(* CoDeSys 2.3.9.42 project: GLX_VCU_v3.3.0.pro *)
(* Author: JvL *)
(* Libraries: ifm_RAWCan\ifm_RAWCan_NT_V020004.lib 7.6.24 16:48:07, ifm_CR0403\ifm_CR0403_V030400.lib 31.5.24 17:04:27, ifm_CANopen\ifm_NetVarLib_NT_V020004.lib 7.6.24 16:46:42, standard.lib 4.10.05 11:14:46, SysLibCallback.lib 7.6.24 16:43:25, 3S_CANOPENNETVAR.LIB 7.6.24 16:46:41, Iecsfc.lib 13.4.06 15:51:28, Util.lib 7.6.24 16:43:26, ifm_CANopen\3S_CANopenManager.lib 7.6.24 16:46:41, ifm_CANopen\3S_CanDrv.lib 7.6.24 16:46:41 *)

(* PLC configuration (modules and I/O channels)
Configuration [LocalConfiguration] node 0, in %IB0 out %QB0 {IFM_PARAM_WORD_TIME = 0}
AT %IB0 [ChInputBool] Input 00 Bit
AT %IB1 [ChInputBool] Input 01 Bit
AT %IB2 [ChInputBool] Input 02 Bit
AT %IB3 [ChInputBool] Input 03 Bit
IGNITION_KEY AT %IB4 [ChInputBool] Input 04 Bit
CHARGER_INPUT AT %IB5 [ChInputBool] Input 05 Bit
BATTERY1_IGNITION AT %IB6 [ChInputBool] Input 06 Bit
BATTERY2_IGNITION AT %IB7 [ChInputBool] Input 07 Bit
ARM_SWITCH AT %IB8 [ChInputBool] Input 08 Bit
KILL_SWITCH AT %IB9 [ChInputBool] Input 09 Bit
HYDRAULIC_SWITCH AT %IB10 [ChInputBool] Input 10 Bit
EM_SWITCH AT %IB11 [ChInputBool] Input 11 Bit
ARM_LED AT %QB0 [ChOutputBool] Output 00 Bit
PRECHARGE_RELAY AT %QB1 [ChOutputBool] Output 01 Bit
AT %QB2 [ChOutputBool] Output 02 Bit
BRAKE_LIGHT AT %QB3 [ChOutputBool] Output 03 Bit
EM_BRAKE AT %QB4 [ChOutputBool] Output 04 Bit
MCU_IGNITION AT %QB5 [ChOutputBool] Output 05 Bit
BATTERY1_RELAY AT %QB6 [ChOutputBool] Output 06 Bit
BATTERY2_RELAY AT %QB7 [ChOutputBool] Output 07 Bit
HORN AT %QB8 [ChOutputBool] Output 08 Bit
BUZZER AT %QB9 [ChOutputBool] Output 09 Bit
CONTACTOR AT %QB10 [ChOutputBool] Output 10 Bit
CHARGING_LED AT %QB11 [ChOutputBool] Output 11 Bit
System Inputs [LocalSystemInputs] node 2, in %IB12 out %QB12
  SUPPLY_VOLTAGE_VBBS AT %IW6 [ChInputWord] Supply voltage VBBS
  SUPPLY_VOLTAGE_VU AT %IW7 [ChInputWord] Supply voltage VU
  SUPPLY_VOLTAGE_VBB1 AT %IW8 [ChInputWord] Supply voltage VBB1
  SUPPLY_VOLTAGE_VBB2 AT %IW9 [ChInputWord] Supply voltage VBB2
  TEMPERATURE AT %IW10 [ChInputInt] Temperature
J1939 Interface [CAN_J1939] node 1, in %IB37 out %QB12
Interface CAN 2 [CAN_BUS] node 1, in %IB37 out %QB12 {STACK_DWORD_S = 0}
  J1939 Interface [CAN_J1939] node 1, in %IB37 out %QB12
*)

(* Global variable list: CanOpen implicit Variables *)
VAR_GLOBAL CONSTANT
	MAX_CTRLINDEX : INT := 0;
END_VAR

(* Global variable list: Global_Variables *)
VAR_GLOBAL
(*BATTERY*)
	BATTERY1_SOC: BYTE;
	BATTERY1_SOH: BYTE;
	BATTERY1_CHARGING: BOOL;
	BATTERY1_POWER: INT;
	BATTERY1_NTC1: BYTE;
	BATTERY1_NTC2: BYTE;
	BATTERY1_CAN_ERROR: BOOL;
	BATTERY1_CAPACITY: INT;
	BATTERY1_TOTAL_CAPACITY: INT;
	BATTERY1_CURRENT: INT;
	BATTERY1_FULLCHARGE_MIN: REAL;

	BATTERY2_SOC: BYTE;
	BATTERY2_SOH: BYTE;
	BATTERY2_CHARGING: BOOL;
	BATTERY2_POWER: INT;
	BATTERY2_NTC1: BYTE;
	BATTERY2_NTC2: BYTE;
	BATTERY2_CAN_ERROR: BOOL;
	BATTERY2_CAPACITY: INT;
	BATTERY2_TOTAL_CAPACITY: INT;
	BATTERY2_CURRENT: INT;
	BATTERY2_FULLCHARGE_MIN: REAL;

(*MCU <> MOTOR*)
	MOTOR_TARGET_RPM: ARRAY [1..6] OF INT;
	MOTOR_IGNITION: ARRAY [1..6] OF BOOL;

	MOTOR_RPM: ARRAY [1..6] OF INT;
	MOTOR_POWER: ARRAY [1..6] OF INT;
	MOTOR_PHASE_CURRENT: ARRAY [1..6] OF WORD;
	MOTOR_TEMPERATURE:ARRAY [1..6] OF BYTE;
	MCU_TEMPERATURE:ARRAY [1..6] OF BYTE;
	MCU_CAN_ERROR: ARRAY [1..6] OF BOOL;

	MOTOR1_FAULT_ARRAY: ARRAY [1..4] OF BYTE;
	MOTOR2_FAULT_ARRAY: ARRAY [1..4] OF BYTE;
	MOTOR6_FAULT_ARRAY: ARRAY [1..4] OF BYTE;
       MOTOR_OBD_ARRAY: ARRAY [1..6] OF WORD;

(*JOYSTICK*)
	LOG_JX: BYTE;
	LOG_JY: BYTE;
	JOY_ERROR: BOOL;
(*IMU*)
	X_ANGLE_BYTE:BYTE;
	Y_ANGLE_BYTE:BYTE;
	NEG_Y: BOOL;
	NEG_X: BOOL;
	Y_MAX_PEAK: BYTE;
	X_MAX_PEAK: BYTE;
	Y_MIN_PEAK: BYTE;
	X_MIN_PEAK: BYTE;
	IMU_CAN_ERROR:BOOL;
	IMU_ALERT: BOOL;
(*DISPLAY TELEMATICS*)
	HIGH_SPEED: BOOL;
	POWER_MODE: BOOL;
	HILL_HOLD: BOOL;
	DISABLE_MCU_CAN: BOOL;
	TRIP_RESET: BOOL;
      	BATTERY_CHARGING:BOOL;
(*MISC*)
	REVERSE: BOOL;
	MCU_BRAKE: BOOL;
(*HYDRAULICS*)
	HYDRAULIC_IGNITION: BOOL;
(*CALCULATIONS*)
	AVG_RPM: INT;
	RANGE_IN_KM: BYTE;
	SPEED: BYTE;

	RUNTIME: DWORD;
	HYDL_UP_TIME:DWORD;
	VEHICLE_UP_TIME: DWORD;
	VEHICLE_UP_TIME_LT: DWORD;

	ODO_KM: WORD;
	ODO_METER: DWORD;

	TRIP_METER: DWORD;
	TRIP_KM: WORD;

	DUMMY: BOOL;
END_VAR
VAR_GLOBAL RETAIN
	Y_MAX_RETAIN: BYTE;
	X_MAX_RETAIN: BYTE;
	Y_MIN_RETAIN: BYTE;
	X_MIN_RETAIN: BYTE;
END_VAR

(* Global variable list: Networkmanagement implicit Variables CAN *)
VAR_GLOBAL CONSTANT
	USE_NWVARS_CAN : BOOL := FALSE;
	MAX_NetVarItems_CAN	: INT := 0;
	MAX_NetVarPDO_Rx_CAN	: INT := 0;
	MAX_NetVarPDO_Tx_CAN	: INT := 0;
	MAX_NetVarOD_CAN		: INT := 0;
END_VAR
VAR_GLOBAL
	pNetVarItems_CAN		: ARRAY[0..MAX_NetVarItems_CAN] OF NetVarDataItem_CAN;
	pNetVarPDO_Rx_CAN		: ARRAY[0..MAX_NetVarPDO_Rx_CAN] OF NetVarPDO_Rx_CAN;
	pNetVarPDO_Tx_CAN		: ARRAY[0..MAX_NetVarPDO_Tx_CAN] OF NetVarPDO_Tx_CAN;
	pNetVarOD_CAN			: ARRAY[0..MAX_NetVarOD_CAN] OF NetVarOD_CAN;
END_VAR

(* POU PLC_PRG, FBD *)
PROGRAM PLC_PRG
VAR
	CONTACTOR_DELAY: TON;
END_VAR
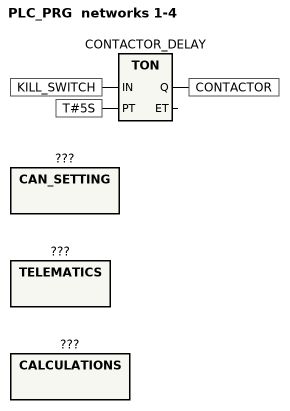
_FBD_ (* Function Block Diagram *)
NETWORK 1
	CONTACTOR_DELAY:TON(IN: KILL_SWITCH, PT: T#5S) => CONTACTOR
NETWORK 2
	???:CAN_SETTING()
NETWORK 3
	???:TELEMATICS()
NETWORK 4
	???:CALCULATIONS()
_END_FBD_
(* the same logic as Structured Text *)
(* Network 1 *)
CONTACTOR_DELAY(IN := KILL_SWITCH, PT := T#5S);
CONTACTOR := CONTACTOR_DELAY.Q;
(* Network 2: see the listing above *)
(* Network 3: see the listing above *)
(* Network 4: see the listing above *)
END_PROGRAM

(* POU CAN_SETTING/CAN_SETTING, FBD *)
PROGRAM CAN_SETTING
(*
Created By: BHAGYESH
Date: 20-01-2024
Version: 1
Description: This program enables the CAN channels and sets the basic CAN parameter for both channels.
This block also controls the IFM's Inbuilt LED.
*)
VAR
	CAN_EN_1: CAN_ENABLE;
	CAN_EN_2: CAN_ENABLE;
	CAN_SET_1: CAN_SETDOWNLOADID;
	CAN_SET_2: CAN_SETDOWNLOADID;
	LED_SET: SET_LED;
	CAN_STATUS_1: CAN_STATUS;
	CAN_STATUS_2: CAN_STATUS;
	RESET_1: BOOL;
	RESET_2: BOOL;
END_VAR
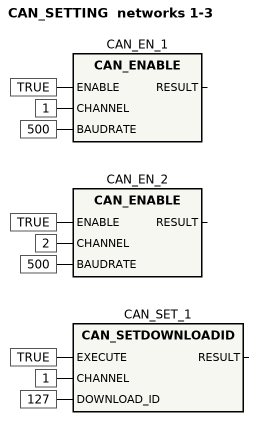
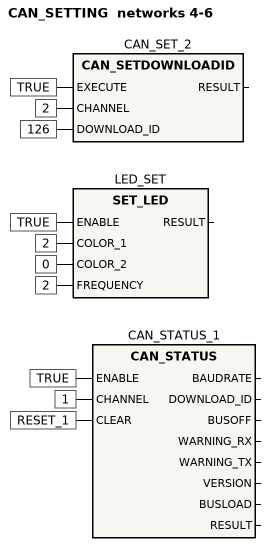
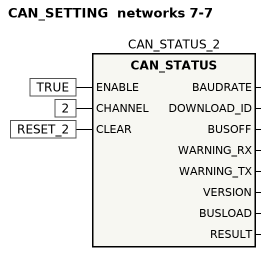
_FBD_ (* Function Block Diagram *)
NETWORK 1
	CAN_EN_1:CAN_ENABLE(ENABLE: TRUE, CHANNEL: 1, BAUDRATE: 500)
NETWORK 2
	CAN_EN_2:CAN_ENABLE(ENABLE: TRUE, CHANNEL: 2, BAUDRATE: 500)
NETWORK 3
	CAN_SET_1:CAN_SETDOWNLOADID(EXECUTE: TRUE, CHANNEL: 1, DOWNLOAD_ID: 127)
NETWORK 4
	CAN_SET_2:CAN_SETDOWNLOADID(EXECUTE: TRUE, CHANNEL: 2, DOWNLOAD_ID: 126)
NETWORK 5
	LED_SET:SET_LED(ENABLE: TRUE, COLOR_1: 2, COLOR_2: 0, FREQUENCY: 2)
NETWORK 6
	CAN_STATUS_1:CAN_STATUS(ENABLE: TRUE, CHANNEL: 1, CLEAR: RESET_1)
NETWORK 7
	CAN_STATUS_2:CAN_STATUS(ENABLE: TRUE, CHANNEL: 2, CLEAR: RESET_2)
_END_FBD_
(* the same logic as Structured Text *)
(* Network 1 *)
CAN_EN_1(ENABLE := TRUE, CHANNEL := 1, BAUDRATE := 500);
(* Network 2 *)
CAN_EN_2(ENABLE := TRUE, CHANNEL := 2, BAUDRATE := 500);
(* Network 3 *)
CAN_SET_1(EXECUTE := TRUE, CHANNEL := 1, DOWNLOAD_ID := 127);
(* Network 4 *)
CAN_SET_2(EXECUTE := TRUE, CHANNEL := 2, DOWNLOAD_ID := 126);
(* Network 5 *)
LED_SET(ENABLE := TRUE, COLOR_1 := 2, COLOR_2 := 0, FREQUENCY := 2);
(* Network 6 *)
CAN_STATUS_1(ENABLE := TRUE, CHANNEL := 1, CLEAR := RESET_1);
(* Network 7 *)
CAN_STATUS_2(ENABLE := TRUE, CHANNEL := 2, CLEAR := RESET_2);
END_PROGRAM

(* POU TELEMATICS, LD *)
PROGRAM TELEMATICS
VAR
	TX_300: CAN_TX;
	TX_301: CAN_TX;
	TX_303: CAN_TX;
	TX_305: CAN_TX;
	TX_306: CAN_TX;
   	TX_307: CAN_TX;
	TX_308: CAN_TX;
	TX_310: CAN_TX;
	TX_311: CAN_TX;
	TX_312: CAN_TX;
	TX_313: CAN_TX;
	TX_31A: CAN_TX;
	TX_31B: CAN_TX;

	TX_400: CAN_TX;
	TX_401: CAN_TX;
	TX_403: CAN_TX;
	TX_405: CAN_TX;
	TX_406: CAN_TX;
   	TX_407: CAN_TX;
	TX_408: CAN_TX;
	TX_410: CAN_TX;
	TX_411: CAN_TX;
	TX_412: CAN_TX;
	TX_413: CAN_TX;
	TX_41A: CAN_TX;
	TX_41B: CAN_TX;
	TX_262: CAN_TX;

	RX_7F0: RX_CAN;
	RX_450: RX_CAN;

	PACK_301: PACK_BYTES;
	PACK_303: PACK_BYTES;
	PACK_305: PACK_BYTES;
	PACK_306: PACK_BYTES;
	PACK_308: PACK_BYTES;
	PACK_311: PACK_BYTES;
	PACK_313: PACK_BYTES;
	PACK_31B: PACK_BYTES;
	PACK_262: PACK_BYTES;

	WB_BATTERY1_POWER: WORD_BYTE_CONVERSION;
	WB_RPM_1: WORD_BYTE_CONVERSION;
	WB_POWER_1: WORD_BYTE_CONVERSION;
	WB_PHASE_1: WORD_BYTE_CONVERSION;
	WB_TARGET_RPM_1: WORD_BYTE_CONVERSION;

	WB_BATTERY2_POWER: WORD_BYTE_CONVERSION;
	WB_RPM_2: WORD_BYTE_CONVERSION;
	WB_POWER_2: WORD_BYTE_CONVERSION;
	WB_PHASE_2: WORD_BYTE_CONVERSION;
	WB_TARGET_RPM_2: WORD_BYTE_CONVERSION;

	WB_RPM_6: WORD_BYTE_CONVERSION;
	WB_POWER_6: WORD_BYTE_CONVERSION;
	WB_PHASE_6: WORD_BYTE_CONVERSION;
	WB_TARGET_RPM_6: WORD_BYTE_CONVERSION;
	WB_FAULTS_6: WORD_BYTE_CONVERSION;

	WB_RUNTIME: WORD_BYTE_CONVERSION;

	DATA_LOG_ERROR: BOOL;
	DWIN_CAN_ERROR: BOOL;
	TIMER_DATALOG: TON;
	TIMER_DWIN: TON;
	TIMER_TX: TON;

	WD_BATTERY1_FULLCHARGE_MIN: WORD;
	WD_BATTERY2_FULLCHARGE_MIN: WORD;
	WB_FULLCHARGE1_MIN: WORD_BYTE_CONVERSION;
	WB_FULLCHARGE2_MIN: WORD_BYTE_CONVERSION;

	WB_OBD_1: WORD_BYTE_CONVERSION;
	WB_OBD_2: WORD_BYTE_CONVERSION;
	WB_OBD_6: WORD_BYTE_CONVERSION;

	WB_HYDL_UP_TIME: WORD_BYTE_CONVERSION;
	WB_TRIP_KM: WORD_BYTE_CONVERSION;
	WB_ODO_METERS: DWORD_BYTE_CONVERSION;
	WB_RUNTIME_MIN: DWORD_BYTE_CONVERSION;
	TIMER_TX_1: TON;
	TIMER_TX_2: TON;
	RX_3A0: RX_CAN;
	TRIP: WORD_BYTE_CONVERSION;
	OBD1_INT: INT;
	OBD1_BYTE: BYTE;
	OBD2_INT: INT;
	OBD2_BYTE: BYTE;
	OBD6_INT: INT;
	OBD6_BYTE: BYTE;
	WB_HYDL_UPTIME: DWORD_BYTE_CONVERSION;
	WB_VEHICLE_UPTIME: DWORD_BYTE_CONVERSION;
	TX_409: CAN_TX;
	PACK_409: PACK_BYTES;
	WB_VEHICLE_UPTIME_LT: DWORD_BYTE_CONVERSION;
END_VAR
VAR CONSTANT
	META_FRAME: ARRAY [0..7] OF BYTE := 18,1,1,0,0,0,0,0; (*GLX_PR, KEY1, VX,VY,VZ*)
	CAN_CHANNEL: BYTE := 1;
END_VAR
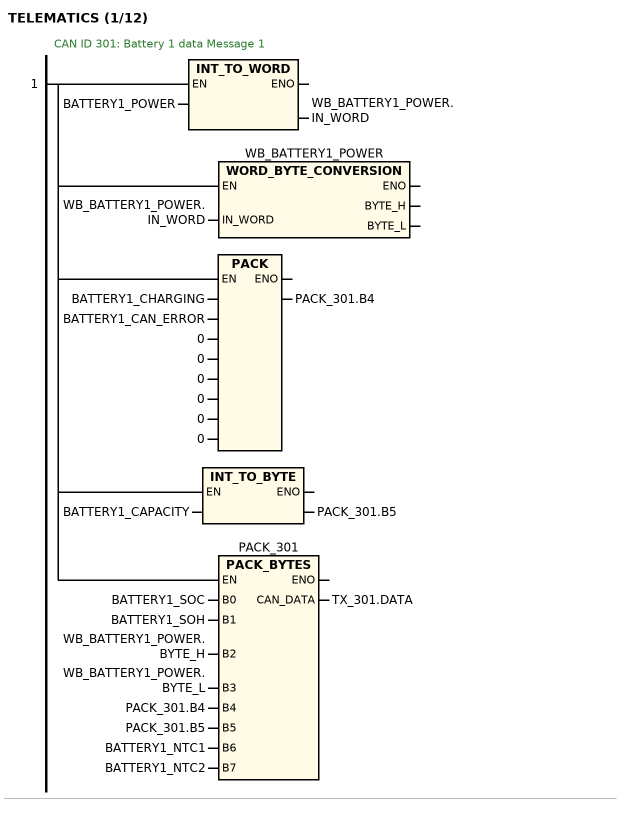
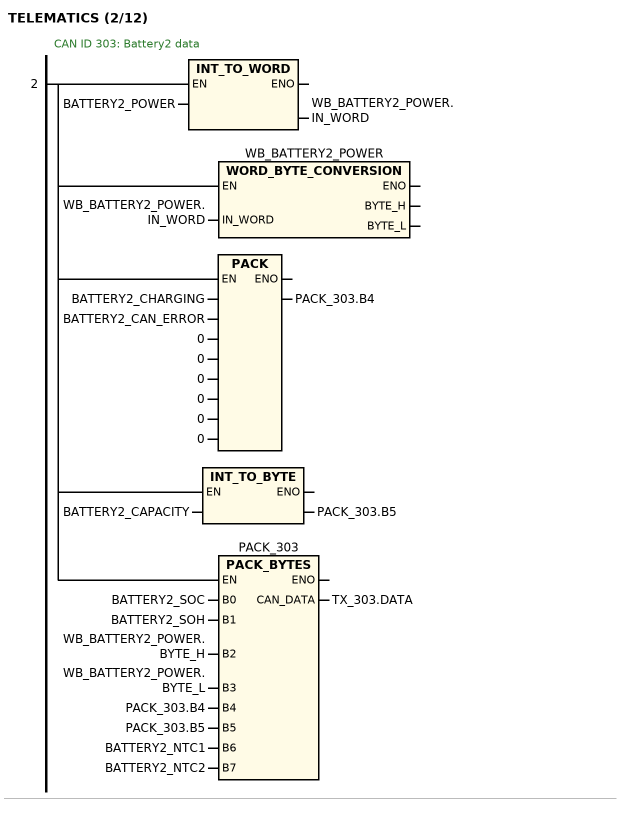
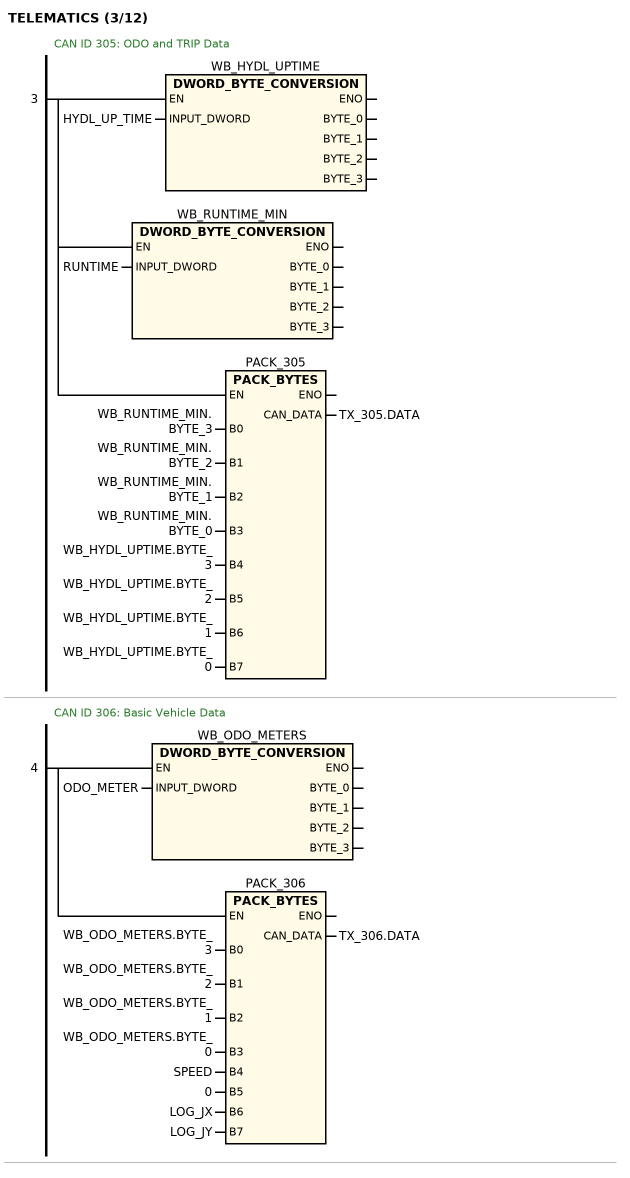
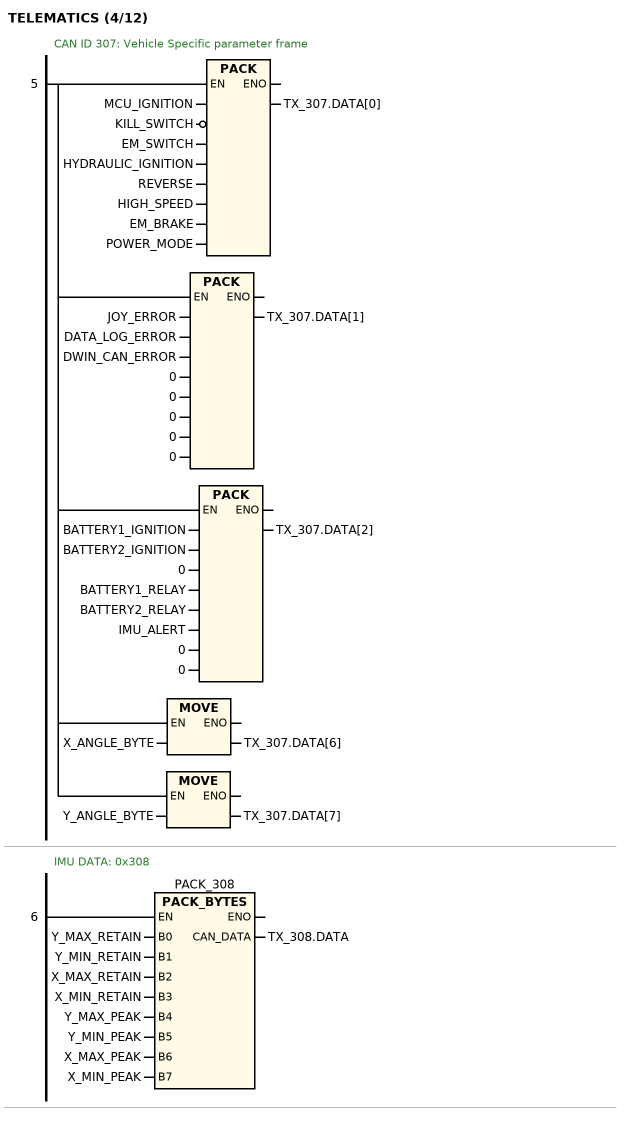
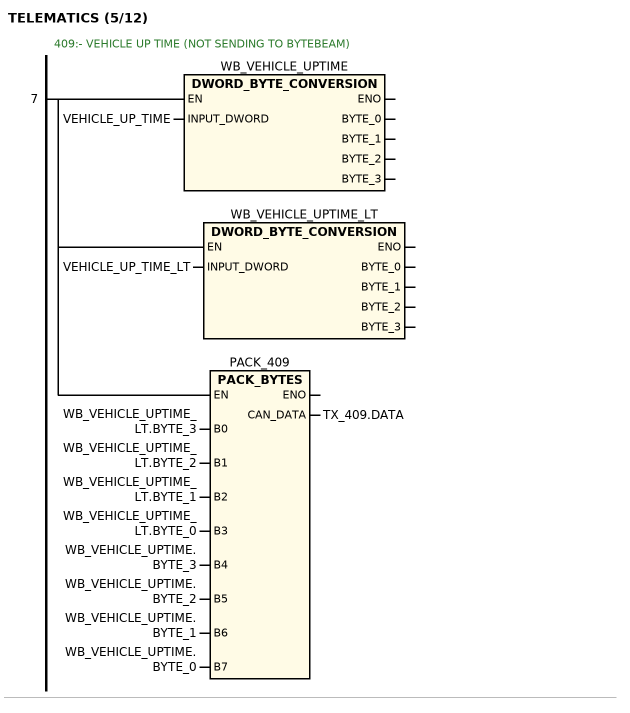
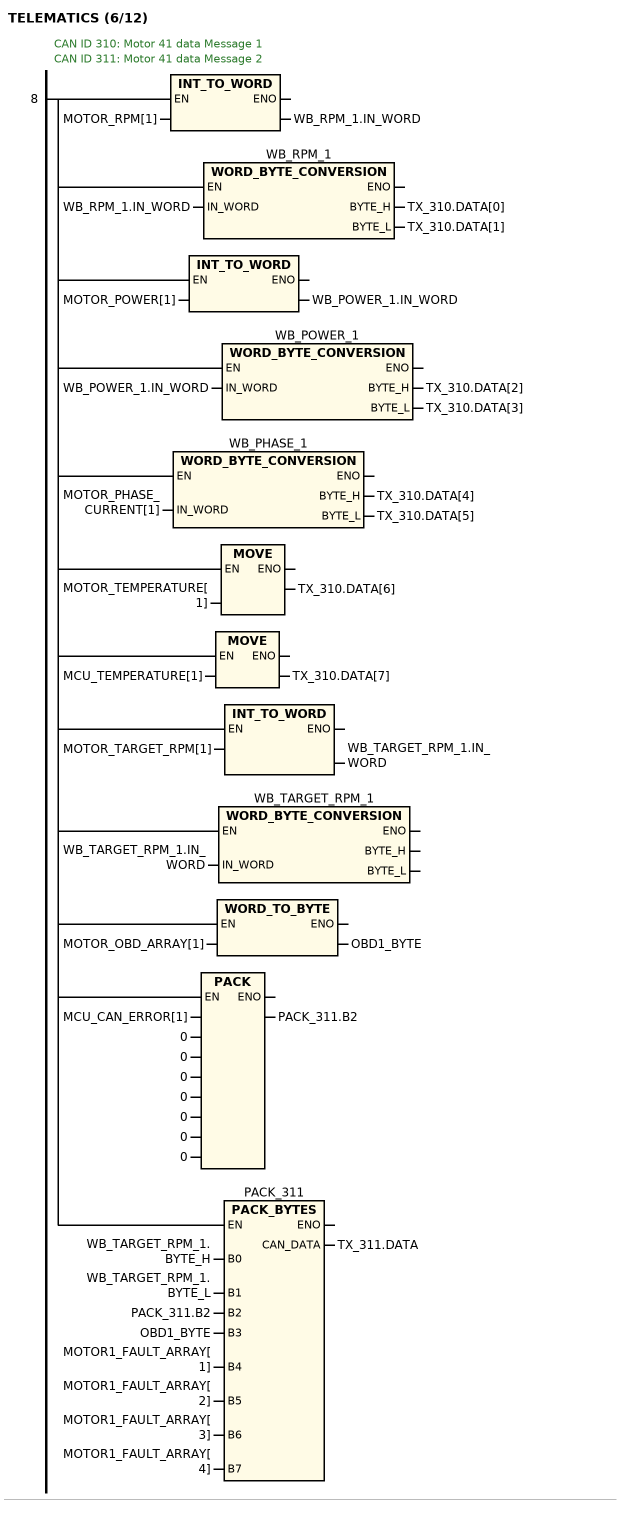
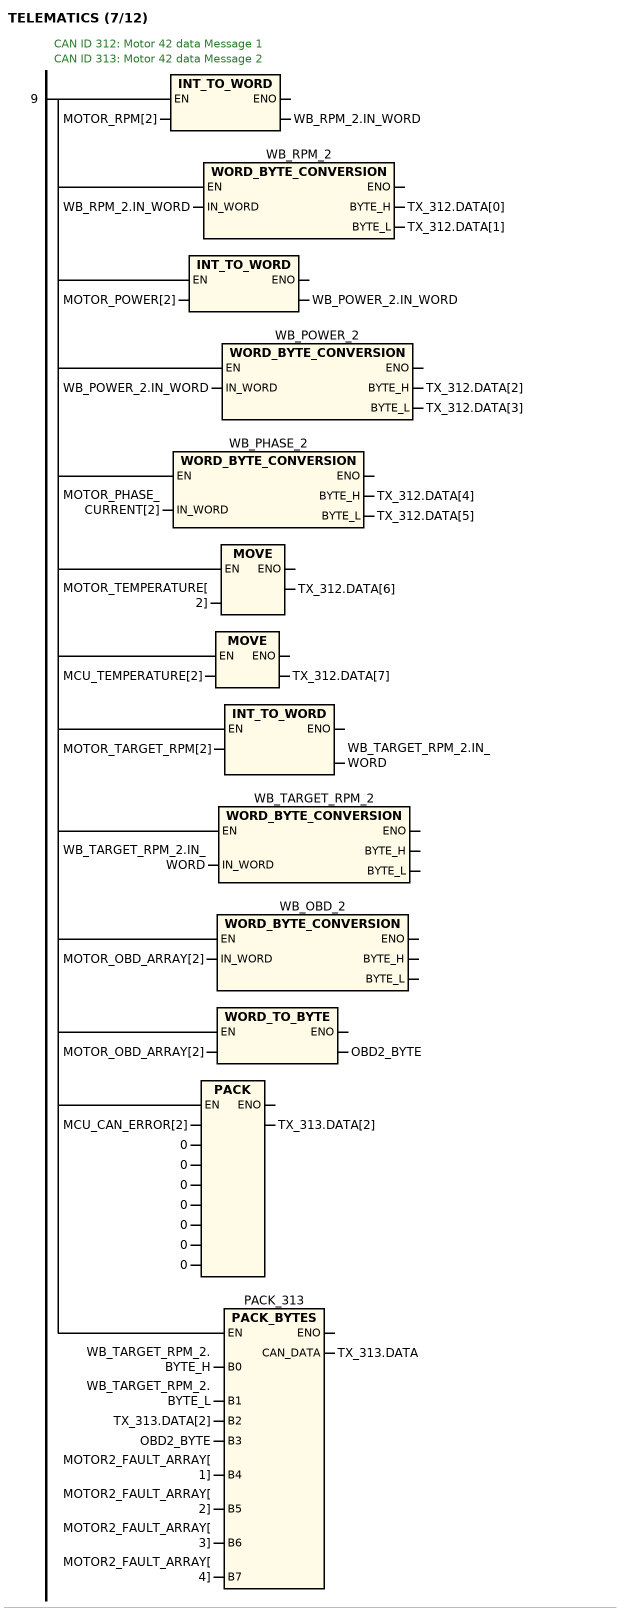
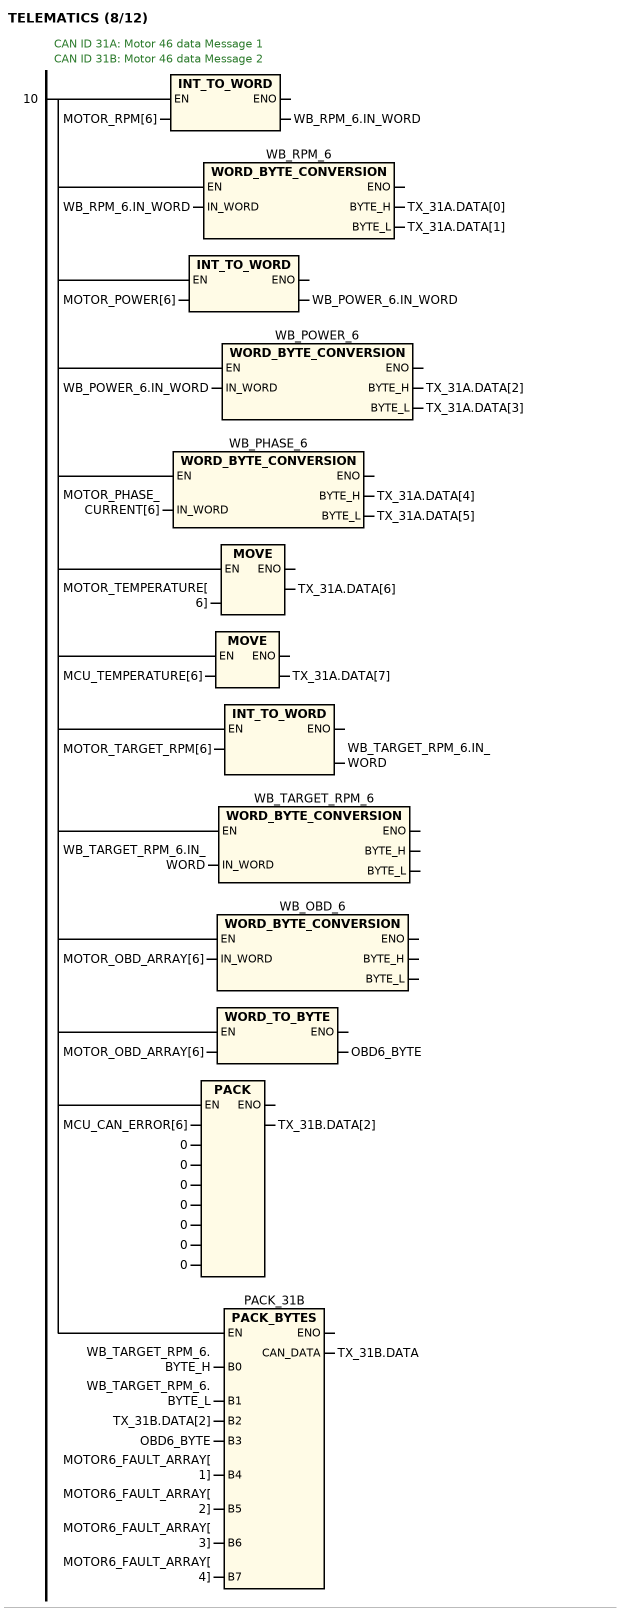
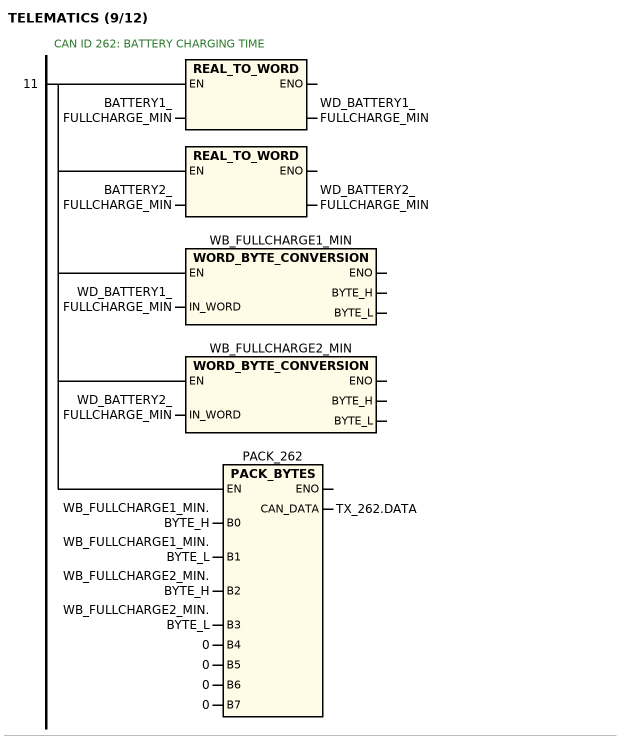
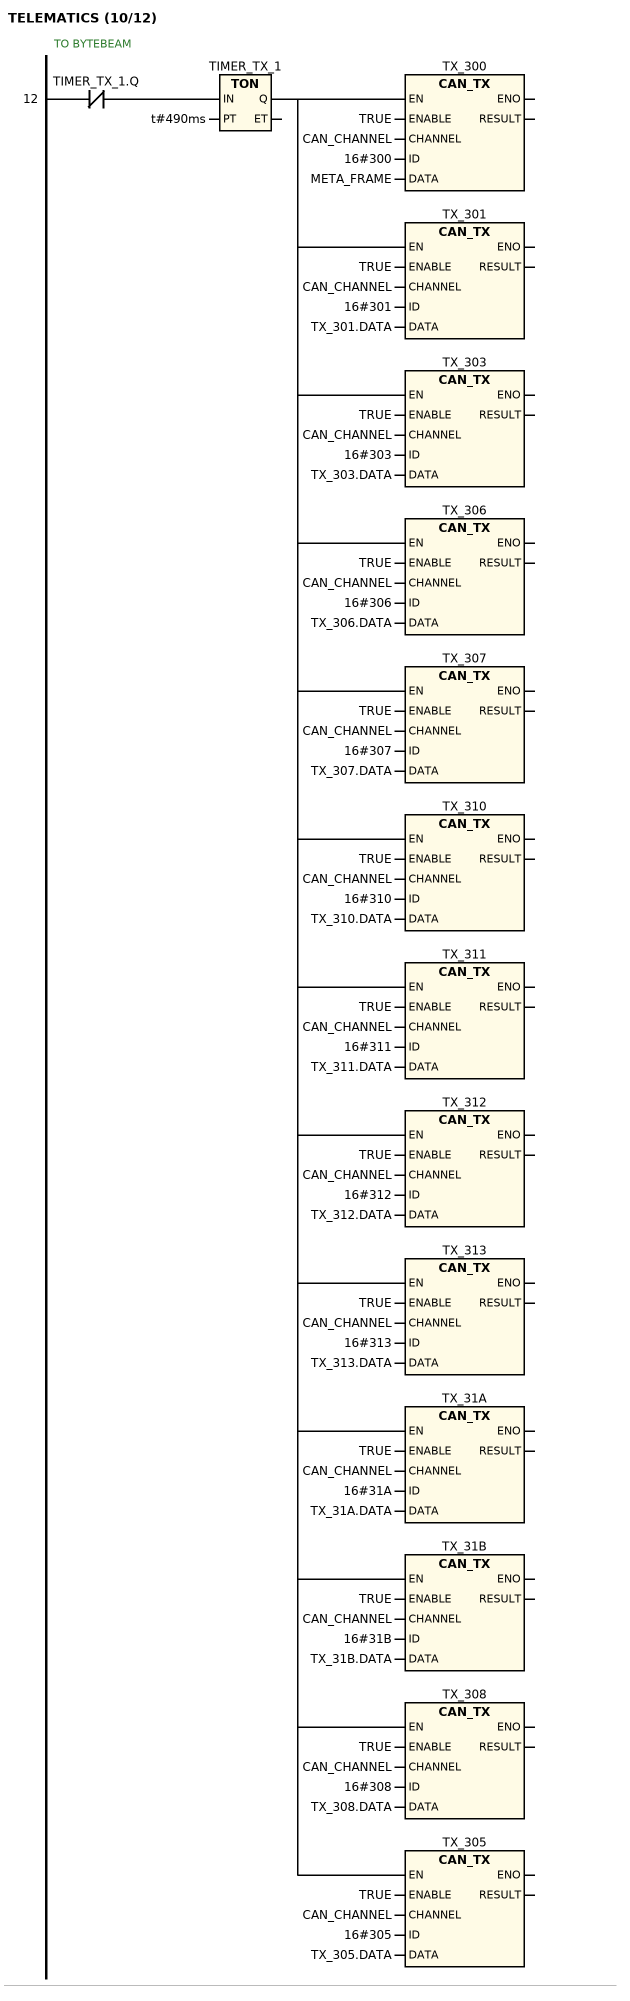
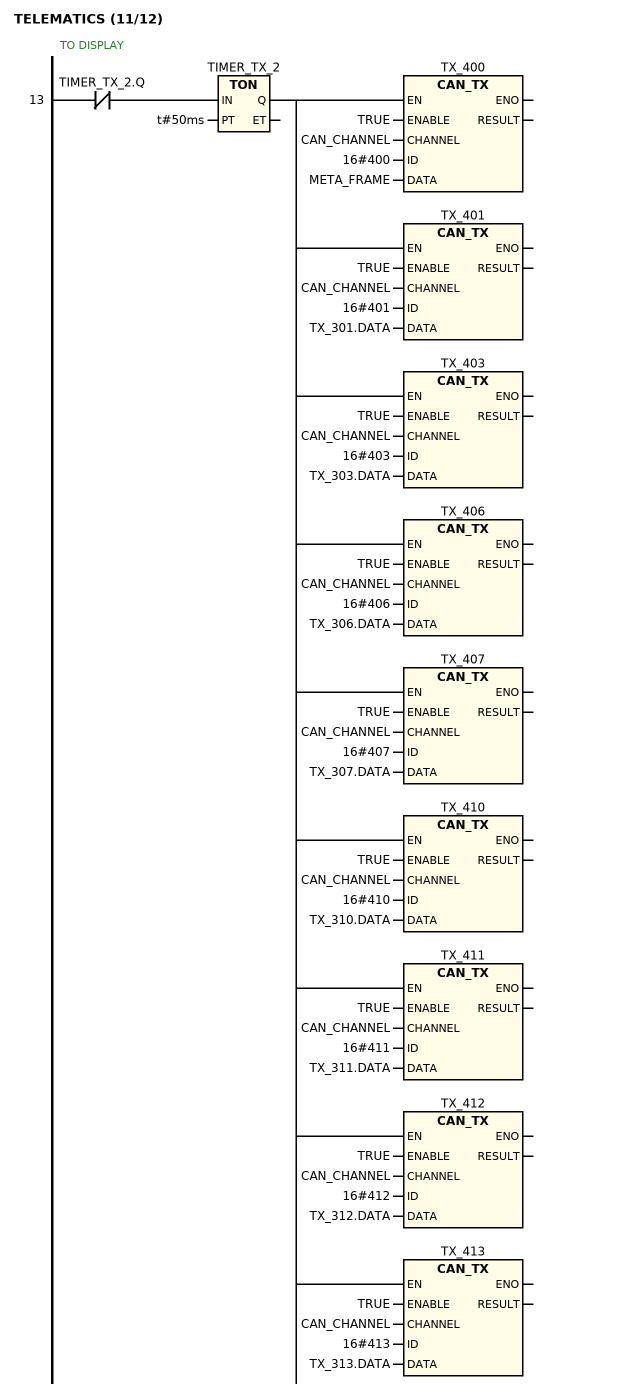
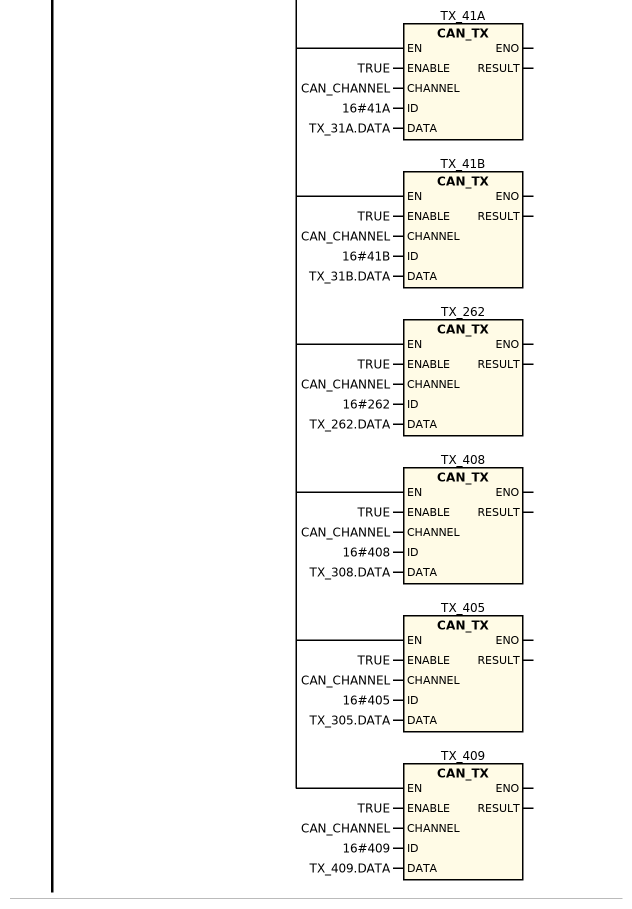
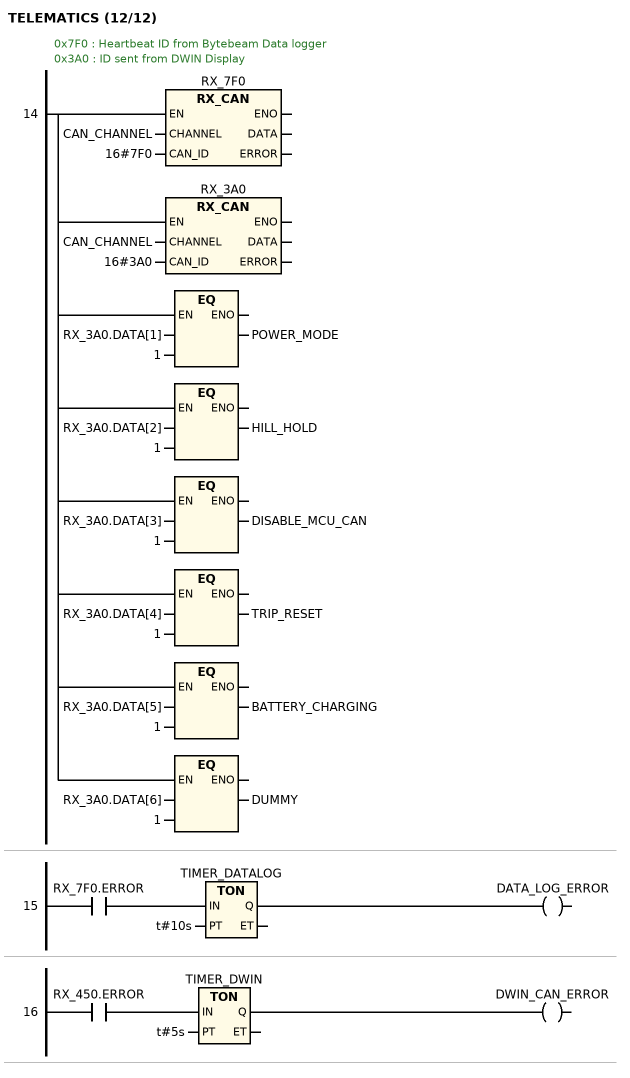
_LD_ (* Ladder Diagram *)
NETWORK 1 (* CAN ID 301: Battery 1 data Message 1 *)
	*
		EN --- INT_TO_WORD(BATTERY1_POWER) => WB_BATTERY1_POWER.IN_WORD
		EN --- WB_BATTERY1_POWER:WORD_BYTE_CONVERSION(IN_WORD: WB_BATTERY1_POWER.IN_WORD)
		EN --- PACK(BATTERY1_CHARGING, BATTERY1_CAN_ERROR, 0, 0, 0, 0, 0, 0) => PACK_301.B4
		EN --- INT_TO_BYTE(BATTERY1_CAPACITY) => PACK_301.B5
		EN --- PACK_301:PACK_BYTES(B0: BATTERY1_SOC, B1: BATTERY1_SOH, B2: WB_BATTERY1_POWER.BYTE_H, B3: WB_BATTERY1_POWER.BYTE_L, B4: PACK_301.B4, B5: PACK_301.B5, B6: BATTERY1_NTC1, B7: BATTERY1_NTC2) => TX_301.DATA
NETWORK 2 (* CAN ID 303: Battery2 data *)
	*
		EN --- INT_TO_WORD(BATTERY2_POWER) => WB_BATTERY2_POWER.IN_WORD
		EN --- WB_BATTERY2_POWER:WORD_BYTE_CONVERSION(IN_WORD: WB_BATTERY2_POWER.IN_WORD)
		EN --- PACK(BATTERY2_CHARGING, BATTERY2_CAN_ERROR, 0, 0, 0, 0, 0, 0) => PACK_303.B4
		EN --- INT_TO_BYTE(BATTERY2_CAPACITY) => PACK_303.B5
		EN --- PACK_303:PACK_BYTES(B0: BATTERY2_SOC, B1: BATTERY2_SOH, B2: WB_BATTERY2_POWER.BYTE_H, B3: WB_BATTERY2_POWER.BYTE_L, B4: PACK_303.B4, B5: PACK_303.B5, B6: BATTERY2_NTC1, B7: BATTERY2_NTC2) => TX_303.DATA
NETWORK 3 (* CAN ID 305: ODO and TRIP Data *)
	*
		EN --- WB_HYDL_UPTIME:DWORD_BYTE_CONVERSION(INPUT_DWORD: HYDL_UP_TIME)
		EN --- WB_RUNTIME_MIN:DWORD_BYTE_CONVERSION(INPUT_DWORD: RUNTIME)
		EN --- PACK_305:PACK_BYTES(B0: WB_RUNTIME_MIN.BYTE_3, B1: WB_RUNTIME_MIN.BYTE_2, B2: WB_RUNTIME_MIN.BYTE_1, B3: WB_RUNTIME_MIN.BYTE_0, B4: WB_HYDL_UPTIME.BYTE_3, B5: WB_HYDL_UPTIME.BYTE_2, B6: WB_HYDL_UPTIME.BYTE_1, B7: WB_HYDL_UPTIME.BYTE_0) => TX_305.DATA
NETWORK 4 (* CAN ID 306: Basic Vehicle Data *)
	*
		EN --- WB_ODO_METERS:DWORD_BYTE_CONVERSION(INPUT_DWORD: ODO_METER)
		EN --- PACK_306:PACK_BYTES(B0: WB_ODO_METERS.BYTE_3, B1: WB_ODO_METERS.BYTE_2, B2: WB_ODO_METERS.BYTE_1, B3: WB_ODO_METERS.BYTE_0, B4: SPEED, B5: 0, B6: LOG_JX, B7: LOG_JY) => TX_306.DATA
NETWORK 5 (* CAN ID 307: Vehicle Specific parameter frame *)
	*
		EN --- PACK(MCU_IGNITION, NOT KILL_SWITCH, EM_SWITCH, HYDRAULIC_IGNITION, REVERSE, HIGH_SPEED, EM_BRAKE, POWER_MODE) => TX_307.DATA[0]
		EN --- PACK(JOY_ERROR, DATA_LOG_ERROR, DWIN_CAN_ERROR, 0, 0, 0, 0, 0) => TX_307.DATA[1]
		EN --- PACK(BATTERY1_IGNITION, BATTERY2_IGNITION, 0, BATTERY1_RELAY, BATTERY2_RELAY, IMU_ALERT, 0, 0) => TX_307.DATA[2]
		EN --- MOVE(X_ANGLE_BYTE) => TX_307.DATA[6]
		EN --- MOVE(Y_ANGLE_BYTE) => TX_307.DATA[7]
NETWORK 6 (* IMU DATA: 0x308 *)
	*
		EN --- PACK_308:PACK_BYTES(B0: Y_MAX_RETAIN, B1: Y_MIN_RETAIN, B2: X_MAX_RETAIN, B3: X_MIN_RETAIN, B4: Y_MAX_PEAK, B5: Y_MIN_PEAK, B6: X_MAX_PEAK, B7: X_MIN_PEAK) => TX_308.DATA
NETWORK 7 (* 409:- VEHICLE UP TIME (NOT SENDING TO BYTEBEAM) *)
	*
		EN --- WB_VEHICLE_UPTIME:DWORD_BYTE_CONVERSION(INPUT_DWORD: VEHICLE_UP_TIME)
		EN --- WB_VEHICLE_UPTIME_LT:DWORD_BYTE_CONVERSION(INPUT_DWORD: VEHICLE_UP_TIME_LT)
		EN --- PACK_409:PACK_BYTES(B0: WB_VEHICLE_UPTIME_LT.BYTE_3, B1: WB_VEHICLE_UPTIME_LT.BYTE_2, B2: WB_VEHICLE_UPTIME_LT.BYTE_1, B3: WB_VEHICLE_UPTIME_LT.BYTE_0, B4: WB_VEHICLE_UPTIME.BYTE_3, B5: WB_VEHICLE_UPTIME.BYTE_2, B6: WB_VEHICLE_UPTIME.BYTE_1, B7: WB_VEHICLE_UPTIME.BYTE_0) => TX_409.DATA
NETWORK 8 (* CAN ID 310: Motor 41 data Message 1 / CAN ID 311: Motor 41 data Message 2 *)
	*
		EN --- INT_TO_WORD(MOTOR_RPM[1]) => WB_RPM_1.IN_WORD
		EN --- WB_RPM_1:WORD_BYTE_CONVERSION(IN_WORD: WB_RPM_1.IN_WORD, BYTE_L => TX_310.DATA[1]) => TX_310.DATA[0]
		EN --- INT_TO_WORD(MOTOR_POWER[1]) => WB_POWER_1.IN_WORD
		EN --- WB_POWER_1:WORD_BYTE_CONVERSION(IN_WORD: WB_POWER_1.IN_WORD, BYTE_L => TX_310.DATA[3]) => TX_310.DATA[2]
		EN --- WB_PHASE_1:WORD_BYTE_CONVERSION(IN_WORD: MOTOR_PHASE_CURRENT[1], BYTE_L => TX_310.DATA[5]) => TX_310.DATA[4]
		EN --- MOVE(MOTOR_TEMPERATURE[1]) => TX_310.DATA[6]
		EN --- MOVE(MCU_TEMPERATURE[1]) => TX_310.DATA[7]
		EN --- INT_TO_WORD(MOTOR_TARGET_RPM[1]) => WB_TARGET_RPM_1.IN_WORD
		EN --- WB_TARGET_RPM_1:WORD_BYTE_CONVERSION(IN_WORD: WB_TARGET_RPM_1.IN_WORD)
		EN --- WORD_TO_BYTE(MOTOR_OBD_ARRAY[1]) => OBD1_BYTE
		EN --- PACK(MCU_CAN_ERROR[1], 0, 0, 0, 0, 0, 0, 0) => PACK_311.B2
		EN --- PACK_311:PACK_BYTES(B0: WB_TARGET_RPM_1.BYTE_H, B1: WB_TARGET_RPM_1.BYTE_L, B2: PACK_311.B2, B3: OBD1_BYTE, B4: MOTOR1_FAULT_ARRAY[1], B5: MOTOR1_FAULT_ARRAY[2], B6: MOTOR1_FAULT_ARRAY[3], B7: MOTOR1_FAULT_ARRAY[4]) => TX_311.DATA
NETWORK 9 (* CAN ID 312: Motor 42 data Message 1 / CAN ID 313: Motor 42 data Message 2 *)
	*
		EN --- INT_TO_WORD(MOTOR_RPM[2]) => WB_RPM_2.IN_WORD
		EN --- WB_RPM_2:WORD_BYTE_CONVERSION(IN_WORD: WB_RPM_2.IN_WORD, BYTE_L => TX_312.DATA[1]) => TX_312.DATA[0]
		EN --- INT_TO_WORD(MOTOR_POWER[2]) => WB_POWER_2.IN_WORD
		EN --- WB_POWER_2:WORD_BYTE_CONVERSION(IN_WORD: WB_POWER_2.IN_WORD, BYTE_L => TX_312.DATA[3]) => TX_312.DATA[2]
		EN --- WB_PHASE_2:WORD_BYTE_CONVERSION(IN_WORD: MOTOR_PHASE_CURRENT[2], BYTE_L => TX_312.DATA[5]) => TX_312.DATA[4]
		EN --- MOVE(MOTOR_TEMPERATURE[2]) => TX_312.DATA[6]
		EN --- MOVE(MCU_TEMPERATURE[2]) => TX_312.DATA[7]
		EN --- INT_TO_WORD(MOTOR_TARGET_RPM[2]) => WB_TARGET_RPM_2.IN_WORD
		EN --- WB_TARGET_RPM_2:WORD_BYTE_CONVERSION(IN_WORD: WB_TARGET_RPM_2.IN_WORD)
		EN --- WB_OBD_2:WORD_BYTE_CONVERSION(IN_WORD: MOTOR_OBD_ARRAY[2])
		EN --- WORD_TO_BYTE(MOTOR_OBD_ARRAY[2]) => OBD2_BYTE
		EN --- PACK(MCU_CAN_ERROR[2], 0, 0, 0, 0, 0, 0, 0) => TX_313.DATA[2]
		EN --- PACK_313:PACK_BYTES(B0: WB_TARGET_RPM_2.BYTE_H, B1: WB_TARGET_RPM_2.BYTE_L, B2: TX_313.DATA[2], B3: OBD2_BYTE, B4: MOTOR2_FAULT_ARRAY[1], B5: MOTOR2_FAULT_ARRAY[2], B6: MOTOR2_FAULT_ARRAY[3], B7: MOTOR2_FAULT_ARRAY[4]) => TX_313.DATA
NETWORK 10 (* CAN ID 31A: Motor 46 data Message 1 / CAN ID 31B: Motor 46 data Message 2 *)
	*
		EN --- INT_TO_WORD(MOTOR_RPM[6]) => WB_RPM_6.IN_WORD
		EN --- WB_RPM_6:WORD_BYTE_CONVERSION(IN_WORD: WB_RPM_6.IN_WORD, BYTE_L => TX_31A.DATA[1]) => TX_31A.DATA[0]
		EN --- INT_TO_WORD(MOTOR_POWER[6]) => WB_POWER_6.IN_WORD
		EN --- WB_POWER_6:WORD_BYTE_CONVERSION(IN_WORD: WB_POWER_6.IN_WORD, BYTE_L => TX_31A.DATA[3]) => TX_31A.DATA[2]
		EN --- WB_PHASE_6:WORD_BYTE_CONVERSION(IN_WORD: MOTOR_PHASE_CURRENT[6], BYTE_L => TX_31A.DATA[5]) => TX_31A.DATA[4]
		EN --- MOVE(MOTOR_TEMPERATURE[6]) => TX_31A.DATA[6]
		EN --- MOVE(MCU_TEMPERATURE[6]) => TX_31A.DATA[7]
		EN --- INT_TO_WORD(MOTOR_TARGET_RPM[6]) => WB_TARGET_RPM_6.IN_WORD
		EN --- WB_TARGET_RPM_6:WORD_BYTE_CONVERSION(IN_WORD: WB_TARGET_RPM_6.IN_WORD)
		EN --- WB_OBD_6:WORD_BYTE_CONVERSION(IN_WORD: MOTOR_OBD_ARRAY[6])
		EN --- WORD_TO_BYTE(MOTOR_OBD_ARRAY[6]) => OBD6_BYTE
		EN --- PACK(MCU_CAN_ERROR[6], 0, 0, 0, 0, 0, 0, 0) => TX_31B.DATA[2]
		EN --- PACK_31B:PACK_BYTES(B0: WB_TARGET_RPM_6.BYTE_H, B1: WB_TARGET_RPM_6.BYTE_L, B2: TX_31B.DATA[2], B3: OBD6_BYTE, B4: MOTOR6_FAULT_ARRAY[1], B5: MOTOR6_FAULT_ARRAY[2], B6: MOTOR6_FAULT_ARRAY[3], B7: MOTOR6_FAULT_ARRAY[4]) => TX_31B.DATA
NETWORK 11 (* CAN ID 262: BATTERY CHARGING TIME *)
	*
		EN --- REAL_TO_WORD(BATTERY1_FULLCHARGE_MIN) => WD_BATTERY1_FULLCHARGE_MIN
		EN --- REAL_TO_WORD(BATTERY2_FULLCHARGE_MIN) => WD_BATTERY2_FULLCHARGE_MIN
		EN --- WB_FULLCHARGE1_MIN:WORD_BYTE_CONVERSION(IN_WORD: WD_BATTERY1_FULLCHARGE_MIN)
		EN --- WB_FULLCHARGE2_MIN:WORD_BYTE_CONVERSION(IN_WORD: WD_BATTERY2_FULLCHARGE_MIN)
		EN --- PACK_262:PACK_BYTES(B0: WB_FULLCHARGE1_MIN.BYTE_H, B1: WB_FULLCHARGE1_MIN.BYTE_L, B2: WB_FULLCHARGE2_MIN.BYTE_H, B3: WB_FULLCHARGE2_MIN.BYTE_L, B4: 0, B5: 0, B6: 0, B7: 0) => TX_262.DATA
NETWORK 12 (* TO BYTEBEAM *)
	[/TIMER_TX_1.Q] - TIMER_TX_1:TON(IN: *, PT: t#490ms)
		EN --- TX_300:CAN_TX(ENABLE: TRUE, CHANNEL: CAN_CHANNEL, ID: 16#300, DATA: META_FRAME)
		EN --- TX_301:CAN_TX(ENABLE: TRUE, CHANNEL: CAN_CHANNEL, ID: 16#301, DATA: TX_301.DATA)
		EN --- TX_303:CAN_TX(ENABLE: TRUE, CHANNEL: CAN_CHANNEL, ID: 16#303, DATA: TX_303.DATA)
		EN --- TX_306:CAN_TX(ENABLE: TRUE, CHANNEL: CAN_CHANNEL, ID: 16#306, DATA: TX_306.DATA)
		EN --- TX_307:CAN_TX(ENABLE: TRUE, CHANNEL: CAN_CHANNEL, ID: 16#307, DATA: TX_307.DATA)
		EN --- TX_310:CAN_TX(ENABLE: TRUE, CHANNEL: CAN_CHANNEL, ID: 16#310, DATA: TX_310.DATA)
		EN --- TX_311:CAN_TX(ENABLE: TRUE, CHANNEL: CAN_CHANNEL, ID: 16#311, DATA: TX_311.DATA)
		EN --- TX_312:CAN_TX(ENABLE: TRUE, CHANNEL: CAN_CHANNEL, ID: 16#312, DATA: TX_312.DATA)
		EN --- TX_313:CAN_TX(ENABLE: TRUE, CHANNEL: CAN_CHANNEL, ID: 16#313, DATA: TX_313.DATA)
		EN --- TX_31A:CAN_TX(ENABLE: TRUE, CHANNEL: CAN_CHANNEL, ID: 16#31A, DATA: TX_31A.DATA)
		EN --- TX_31B:CAN_TX(ENABLE: TRUE, CHANNEL: CAN_CHANNEL, ID: 16#31B, DATA: TX_31B.DATA)
		EN --- TX_308:CAN_TX(ENABLE: TRUE, CHANNEL: CAN_CHANNEL, ID: 16#308, DATA: TX_308.DATA)
		EN --- TX_305:CAN_TX(ENABLE: TRUE, CHANNEL: CAN_CHANNEL, ID: 16#305, DATA: TX_305.DATA)
NETWORK 13 (* TO DISPLAY *)
	[/TIMER_TX_2.Q] - TIMER_TX_2:TON(IN: *, PT: t#50ms)
		EN --- TX_400:CAN_TX(ENABLE: TRUE, CHANNEL: CAN_CHANNEL, ID: 16#400, DATA: META_FRAME)
		EN --- TX_401:CAN_TX(ENABLE: TRUE, CHANNEL: CAN_CHANNEL, ID: 16#401, DATA: TX_301.DATA)
		EN --- TX_403:CAN_TX(ENABLE: TRUE, CHANNEL: CAN_CHANNEL, ID: 16#403, DATA: TX_303.DATA)
		EN --- TX_406:CAN_TX(ENABLE: TRUE, CHANNEL: CAN_CHANNEL, ID: 16#406, DATA: TX_306.DATA)
		EN --- TX_407:CAN_TX(ENABLE: TRUE, CHANNEL: CAN_CHANNEL, ID: 16#407, DATA: TX_307.DATA)
		EN --- TX_410:CAN_TX(ENABLE: TRUE, CHANNEL: CAN_CHANNEL, ID: 16#410, DATA: TX_310.DATA)
		EN --- TX_411:CAN_TX(ENABLE: TRUE, CHANNEL: CAN_CHANNEL, ID: 16#411, DATA: TX_311.DATA)
		EN --- TX_412:CAN_TX(ENABLE: TRUE, CHANNEL: CAN_CHANNEL, ID: 16#412, DATA: TX_312.DATA)
		EN --- TX_413:CAN_TX(ENABLE: TRUE, CHANNEL: CAN_CHANNEL, ID: 16#413, DATA: TX_313.DATA)
		EN --- TX_41A:CAN_TX(ENABLE: TRUE, CHANNEL: CAN_CHANNEL, ID: 16#41A, DATA: TX_31A.DATA)
		EN --- TX_41B:CAN_TX(ENABLE: TRUE, CHANNEL: CAN_CHANNEL, ID: 16#41B, DATA: TX_31B.DATA)
		EN --- TX_262:CAN_TX(ENABLE: TRUE, CHANNEL: CAN_CHANNEL, ID: 16#262, DATA: TX_262.DATA)
		EN --- TX_408:CAN_TX(ENABLE: TRUE, CHANNEL: CAN_CHANNEL, ID: 16#408, DATA: TX_308.DATA)
		EN --- TX_405:CAN_TX(ENABLE: TRUE, CHANNEL: CAN_CHANNEL, ID: 16#405, DATA: TX_305.DATA)
		EN --- TX_409:CAN_TX(ENABLE: TRUE, CHANNEL: CAN_CHANNEL, ID: 16#409, DATA: TX_409.DATA)
NETWORK 14 (* 0x7F0 : Heartbeat ID from Bytebeam Data logger / 0x3A0 : ID sent from DWIN Display *)
	*
		EN --- RX_7F0:RX_CAN(CHANNEL: CAN_CHANNEL, CAN_ID: 16#7F0)
		EN --- RX_3A0:RX_CAN(CHANNEL: CAN_CHANNEL, CAN_ID: 16#3A0)
		EN --- EQ(RX_3A0.DATA[1], 1) => POWER_MODE
		EN --- EQ(RX_3A0.DATA[2], 1) => HILL_HOLD
		EN --- EQ(RX_3A0.DATA[3], 1) => DISABLE_MCU_CAN
		EN --- EQ(RX_3A0.DATA[4], 1) => TRIP_RESET
		EN --- EQ(RX_3A0.DATA[5], 1) => BATTERY_CHARGING
		EN --- EQ(RX_3A0.DATA[6], 1) => DUMMY
NETWORK 15
	[RX_7F0.ERROR] - TIMER_DATALOG:TON(IN: *, PT: t#10s) --- (DATA_LOG_ERROR)
NETWORK 16
	[RX_450.ERROR] - TIMER_DWIN:TON(IN: *, PT: t#5s) --- (DWIN_CAN_ERROR)
_END_LD_
(* the same logic as Structured Text *)
(* Network 1: CAN ID 301: Battery 1 data Message 1 *)
WB_BATTERY1_POWER.IN_WORD := INT_TO_WORD(BATTERY1_POWER);
WB_BATTERY1_POWER(IN_WORD := WB_BATTERY1_POWER.IN_WORD);
PACK_301.B4 := PACK(BATTERY1_CHARGING, BATTERY1_CAN_ERROR, 0, 0, 0, 0, 0, 0);
PACK_301.B5 := INT_TO_BYTE(BATTERY1_CAPACITY);
PACK_301(B0 := BATTERY1_SOC, B1 := BATTERY1_SOH, B2 := WB_BATTERY1_POWER.BYTE_H, B3 := WB_BATTERY1_POWER.BYTE_L, B4 := PACK_301.B4, B5 := PACK_301.B5, B6 := BATTERY1_NTC1, B7 := BATTERY1_NTC2);
TX_301.DATA := PACK_301.CAN_DATA;
(* Network 2: CAN ID 303: Battery2 data *)
WB_BATTERY2_POWER.IN_WORD := INT_TO_WORD(BATTERY2_POWER);
WB_BATTERY2_POWER(IN_WORD := WB_BATTERY2_POWER.IN_WORD);
PACK_303.B4 := PACK(BATTERY2_CHARGING, BATTERY2_CAN_ERROR, 0, 0, 0, 0, 0, 0);
PACK_303.B5 := INT_TO_BYTE(BATTERY2_CAPACITY);
PACK_303(B0 := BATTERY2_SOC, B1 := BATTERY2_SOH, B2 := WB_BATTERY2_POWER.BYTE_H, B3 := WB_BATTERY2_POWER.BYTE_L, B4 := PACK_303.B4, B5 := PACK_303.B5, B6 := BATTERY2_NTC1, B7 := BATTERY2_NTC2);
TX_303.DATA := PACK_303.CAN_DATA;
(* Network 3: CAN ID 305: ODO and TRIP Data *)
WB_HYDL_UPTIME(INPUT_DWORD := HYDL_UP_TIME);
WB_RUNTIME_MIN(INPUT_DWORD := RUNTIME);
PACK_305(B0 := WB_RUNTIME_MIN.BYTE_3, B1 := WB_RUNTIME_MIN.BYTE_2, B2 := WB_RUNTIME_MIN.BYTE_1, B3 := WB_RUNTIME_MIN.BYTE_0, B4 := WB_HYDL_UPTIME.BYTE_3, B5 := WB_HYDL_UPTIME.BYTE_2, B6 := WB_HYDL_UPTIME.BYTE_1, B7 := WB_HYDL_UPTIME.BYTE_0);
TX_305.DATA := PACK_305.CAN_DATA;
(* Network 4: CAN ID 306: Basic Vehicle Data *)
WB_ODO_METERS(INPUT_DWORD := ODO_METER);
PACK_306(B0 := WB_ODO_METERS.BYTE_3, B1 := WB_ODO_METERS.BYTE_2, B2 := WB_ODO_METERS.BYTE_1, B3 := WB_ODO_METERS.BYTE_0, B4 := SPEED, B5 := 0, B6 := LOG_JX, B7 := LOG_JY);
TX_306.DATA := PACK_306.CAN_DATA;
(* Network 5: CAN ID 307: Vehicle Specific parameter frame *)
TX_307.DATA[0] := PACK(MCU_IGNITION, NOT KILL_SWITCH, EM_SWITCH, HYDRAULIC_IGNITION, REVERSE, HIGH_SPEED, EM_BRAKE, POWER_MODE);
TX_307.DATA[1] := PACK(JOY_ERROR, DATA_LOG_ERROR, DWIN_CAN_ERROR, 0, 0, 0, 0, 0);
TX_307.DATA[2] := PACK(BATTERY1_IGNITION, BATTERY2_IGNITION, 0, BATTERY1_RELAY, BATTERY2_RELAY, IMU_ALERT, 0, 0);
TX_307.DATA[6] := X_ANGLE_BYTE;
TX_307.DATA[7] := Y_ANGLE_BYTE;
(* Network 6: IMU DATA: 0x308 *)
PACK_308(B0 := Y_MAX_RETAIN, B1 := Y_MIN_RETAIN, B2 := X_MAX_RETAIN, B3 := X_MIN_RETAIN, B4 := Y_MAX_PEAK, B5 := Y_MIN_PEAK, B6 := X_MAX_PEAK, B7 := X_MIN_PEAK);
TX_308.DATA := PACK_308.CAN_DATA;
(* Network 7: 409:- VEHICLE UP TIME (NOT SENDING TO BYTEBEAM) *)
WB_VEHICLE_UPTIME(INPUT_DWORD := VEHICLE_UP_TIME);
WB_VEHICLE_UPTIME_LT(INPUT_DWORD := VEHICLE_UP_TIME_LT);
PACK_409(B0 := WB_VEHICLE_UPTIME_LT.BYTE_3, B1 := WB_VEHICLE_UPTIME_LT.BYTE_2, B2 := WB_VEHICLE_UPTIME_LT.BYTE_1, B3 := WB_VEHICLE_UPTIME_LT.BYTE_0, B4 := WB_VEHICLE_UPTIME.BYTE_3, B5 := WB_VEHICLE_UPTIME.BYTE_2, B6 := WB_VEHICLE_UPTIME.BYTE_1, B7 := WB_VEHICLE_UPTIME.BYTE_0);
TX_409.DATA := PACK_409.CAN_DATA;
(* Network 8: CAN ID 310: Motor 41 data Message 1 / CAN ID 311: Motor 41 data Message 2 *)
WB_RPM_1.IN_WORD := INT_TO_WORD(MOTOR_RPM[1]);
WB_RPM_1(IN_WORD := WB_RPM_1.IN_WORD);
TX_310.DATA[1] := WB_RPM_1.BYTE_L;
TX_310.DATA[0] := WB_RPM_1.BYTE_H;
WB_POWER_1.IN_WORD := INT_TO_WORD(MOTOR_POWER[1]);
WB_POWER_1(IN_WORD := WB_POWER_1.IN_WORD);
TX_310.DATA[3] := WB_POWER_1.BYTE_L;
TX_310.DATA[2] := WB_POWER_1.BYTE_H;
WB_PHASE_1(IN_WORD := MOTOR_PHASE_CURRENT[1]);
TX_310.DATA[5] := WB_PHASE_1.BYTE_L;
TX_310.DATA[4] := WB_PHASE_1.BYTE_H;
TX_310.DATA[6] := MOTOR_TEMPERATURE[1];
TX_310.DATA[7] := MCU_TEMPERATURE[1];
WB_TARGET_RPM_1.IN_WORD := INT_TO_WORD(MOTOR_TARGET_RPM[1]);
WB_TARGET_RPM_1(IN_WORD := WB_TARGET_RPM_1.IN_WORD);
OBD1_BYTE := WORD_TO_BYTE(MOTOR_OBD_ARRAY[1]);
PACK_311.B2 := PACK(MCU_CAN_ERROR[1], 0, 0, 0, 0, 0, 0, 0);
PACK_311(B0 := WB_TARGET_RPM_1.BYTE_H, B1 := WB_TARGET_RPM_1.BYTE_L, B2 := PACK_311.B2, B3 := OBD1_BYTE, B4 := MOTOR1_FAULT_ARRAY[1], B5 := MOTOR1_FAULT_ARRAY[2], B6 := MOTOR1_FAULT_ARRAY[3], B7 := MOTOR1_FAULT_ARRAY[4]);
TX_311.DATA := PACK_311.CAN_DATA;
(* Network 9: CAN ID 312: Motor 42 data Message 1 / CAN ID 313: Motor 42 data Message 2 *)
WB_RPM_2.IN_WORD := INT_TO_WORD(MOTOR_RPM[2]);
WB_RPM_2(IN_WORD := WB_RPM_2.IN_WORD);
TX_312.DATA[1] := WB_RPM_2.BYTE_L;
TX_312.DATA[0] := WB_RPM_2.BYTE_H;
WB_POWER_2.IN_WORD := INT_TO_WORD(MOTOR_POWER[2]);
WB_POWER_2(IN_WORD := WB_POWER_2.IN_WORD);
TX_312.DATA[3] := WB_POWER_2.BYTE_L;
TX_312.DATA[2] := WB_POWER_2.BYTE_H;
WB_PHASE_2(IN_WORD := MOTOR_PHASE_CURRENT[2]);
TX_312.DATA[5] := WB_PHASE_2.BYTE_L;
TX_312.DATA[4] := WB_PHASE_2.BYTE_H;
TX_312.DATA[6] := MOTOR_TEMPERATURE[2];
TX_312.DATA[7] := MCU_TEMPERATURE[2];
WB_TARGET_RPM_2.IN_WORD := INT_TO_WORD(MOTOR_TARGET_RPM[2]);
WB_TARGET_RPM_2(IN_WORD := WB_TARGET_RPM_2.IN_WORD);
WB_OBD_2(IN_WORD := MOTOR_OBD_ARRAY[2]);
OBD2_BYTE := WORD_TO_BYTE(MOTOR_OBD_ARRAY[2]);
TX_313.DATA[2] := PACK(MCU_CAN_ERROR[2], 0, 0, 0, 0, 0, 0, 0);
PACK_313(B0 := WB_TARGET_RPM_2.BYTE_H, B1 := WB_TARGET_RPM_2.BYTE_L, B2 := TX_313.DATA[2], B3 := OBD2_BYTE, B4 := MOTOR2_FAULT_ARRAY[1], B5 := MOTOR2_FAULT_ARRAY[2], B6 := MOTOR2_FAULT_ARRAY[3], B7 := MOTOR2_FAULT_ARRAY[4]);
TX_313.DATA := PACK_313.CAN_DATA;
(* Network 10: CAN ID 31A: Motor 46 data Message 1 / CAN ID 31B: Motor 46 data Message 2 *)
WB_RPM_6.IN_WORD := INT_TO_WORD(MOTOR_RPM[6]);
WB_RPM_6(IN_WORD := WB_RPM_6.IN_WORD);
TX_31A.DATA[1] := WB_RPM_6.BYTE_L;
TX_31A.DATA[0] := WB_RPM_6.BYTE_H;
WB_POWER_6.IN_WORD := INT_TO_WORD(MOTOR_POWER[6]);
WB_POWER_6(IN_WORD := WB_POWER_6.IN_WORD);
TX_31A.DATA[3] := WB_POWER_6.BYTE_L;
TX_31A.DATA[2] := WB_POWER_6.BYTE_H;
WB_PHASE_6(IN_WORD := MOTOR_PHASE_CURRENT[6]);
TX_31A.DATA[5] := WB_PHASE_6.BYTE_L;
TX_31A.DATA[4] := WB_PHASE_6.BYTE_H;
TX_31A.DATA[6] := MOTOR_TEMPERATURE[6];
TX_31A.DATA[7] := MCU_TEMPERATURE[6];
WB_TARGET_RPM_6.IN_WORD := INT_TO_WORD(MOTOR_TARGET_RPM[6]);
WB_TARGET_RPM_6(IN_WORD := WB_TARGET_RPM_6.IN_WORD);
WB_OBD_6(IN_WORD := MOTOR_OBD_ARRAY[6]);
OBD6_BYTE := WORD_TO_BYTE(MOTOR_OBD_ARRAY[6]);
TX_31B.DATA[2] := PACK(MCU_CAN_ERROR[6], 0, 0, 0, 0, 0, 0, 0);
PACK_31B(B0 := WB_TARGET_RPM_6.BYTE_H, B1 := WB_TARGET_RPM_6.BYTE_L, B2 := TX_31B.DATA[2], B3 := OBD6_BYTE, B4 := MOTOR6_FAULT_ARRAY[1], B5 := MOTOR6_FAULT_ARRAY[2], B6 := MOTOR6_FAULT_ARRAY[3], B7 := MOTOR6_FAULT_ARRAY[4]);
TX_31B.DATA := PACK_31B.CAN_DATA;
(* Network 11: CAN ID 262: BATTERY CHARGING TIME *)
WD_BATTERY1_FULLCHARGE_MIN := REAL_TO_WORD(BATTERY1_FULLCHARGE_MIN);
WD_BATTERY2_FULLCHARGE_MIN := REAL_TO_WORD(BATTERY2_FULLCHARGE_MIN);
WB_FULLCHARGE1_MIN(IN_WORD := WD_BATTERY1_FULLCHARGE_MIN);
WB_FULLCHARGE2_MIN(IN_WORD := WD_BATTERY2_FULLCHARGE_MIN);
PACK_262(B0 := WB_FULLCHARGE1_MIN.BYTE_H, B1 := WB_FULLCHARGE1_MIN.BYTE_L, B2 := WB_FULLCHARGE2_MIN.BYTE_H, B3 := WB_FULLCHARGE2_MIN.BYTE_L, B4 := 0, B5 := 0, B6 := 0, B7 := 0);
TX_262.DATA := PACK_262.CAN_DATA;
(* Network 12: TO BYTEBEAM *)
TIMER_TX_1(IN := NOT TIMER_TX_1.Q, PT := t#490ms);
IF TIMER_TX_1.Q THEN
	TX_300(ENABLE := TRUE, CHANNEL := CAN_CHANNEL, ID := 16#300, DATA := META_FRAME);
	TX_301(ENABLE := TRUE, CHANNEL := CAN_CHANNEL, ID := 16#301, DATA := TX_301.DATA);
	TX_303(ENABLE := TRUE, CHANNEL := CAN_CHANNEL, ID := 16#303, DATA := TX_303.DATA);
	TX_306(ENABLE := TRUE, CHANNEL := CAN_CHANNEL, ID := 16#306, DATA := TX_306.DATA);
	TX_307(ENABLE := TRUE, CHANNEL := CAN_CHANNEL, ID := 16#307, DATA := TX_307.DATA);
	TX_310(ENABLE := TRUE, CHANNEL := CAN_CHANNEL, ID := 16#310, DATA := TX_310.DATA);
	TX_311(ENABLE := TRUE, CHANNEL := CAN_CHANNEL, ID := 16#311, DATA := TX_311.DATA);
	TX_312(ENABLE := TRUE, CHANNEL := CAN_CHANNEL, ID := 16#312, DATA := TX_312.DATA);
	TX_313(ENABLE := TRUE, CHANNEL := CAN_CHANNEL, ID := 16#313, DATA := TX_313.DATA);
	TX_31A(ENABLE := TRUE, CHANNEL := CAN_CHANNEL, ID := 16#31A, DATA := TX_31A.DATA);
	TX_31B(ENABLE := TRUE, CHANNEL := CAN_CHANNEL, ID := 16#31B, DATA := TX_31B.DATA);
	TX_308(ENABLE := TRUE, CHANNEL := CAN_CHANNEL, ID := 16#308, DATA := TX_308.DATA);
	TX_305(ENABLE := TRUE, CHANNEL := CAN_CHANNEL, ID := 16#305, DATA := TX_305.DATA);
END_IF;
(* Network 13: TO DISPLAY *)
TIMER_TX_2(IN := NOT TIMER_TX_2.Q, PT := t#50ms);
IF TIMER_TX_2.Q THEN
	TX_400(ENABLE := TRUE, CHANNEL := CAN_CHANNEL, ID := 16#400, DATA := META_FRAME);
	TX_401(ENABLE := TRUE, CHANNEL := CAN_CHANNEL, ID := 16#401, DATA := TX_301.DATA);
	TX_403(ENABLE := TRUE, CHANNEL := CAN_CHANNEL, ID := 16#403, DATA := TX_303.DATA);
	TX_406(ENABLE := TRUE, CHANNEL := CAN_CHANNEL, ID := 16#406, DATA := TX_306.DATA);
	TX_407(ENABLE := TRUE, CHANNEL := CAN_CHANNEL, ID := 16#407, DATA := TX_307.DATA);
	TX_410(ENABLE := TRUE, CHANNEL := CAN_CHANNEL, ID := 16#410, DATA := TX_310.DATA);
	TX_411(ENABLE := TRUE, CHANNEL := CAN_CHANNEL, ID := 16#411, DATA := TX_311.DATA);
	TX_412(ENABLE := TRUE, CHANNEL := CAN_CHANNEL, ID := 16#412, DATA := TX_312.DATA);
	TX_413(ENABLE := TRUE, CHANNEL := CAN_CHANNEL, ID := 16#413, DATA := TX_313.DATA);
	TX_41A(ENABLE := TRUE, CHANNEL := CAN_CHANNEL, ID := 16#41A, DATA := TX_31A.DATA);
	TX_41B(ENABLE := TRUE, CHANNEL := CAN_CHANNEL, ID := 16#41B, DATA := TX_31B.DATA);
	TX_262(ENABLE := TRUE, CHANNEL := CAN_CHANNEL, ID := 16#262, DATA := TX_262.DATA);
	TX_408(ENABLE := TRUE, CHANNEL := CAN_CHANNEL, ID := 16#408, DATA := TX_308.DATA);
	TX_405(ENABLE := TRUE, CHANNEL := CAN_CHANNEL, ID := 16#405, DATA := TX_305.DATA);
	TX_409(ENABLE := TRUE, CHANNEL := CAN_CHANNEL, ID := 16#409, DATA := TX_409.DATA);
END_IF;
(* Network 14: 0x7F0 : Heartbeat ID from Bytebeam Data logger / 0x3A0 : ID sent from DWIN Display *)
RX_7F0(CHANNEL := CAN_CHANNEL, CAN_ID := 16#7F0);
RX_3A0(CHANNEL := CAN_CHANNEL, CAN_ID := 16#3A0);
POWER_MODE := RX_3A0.DATA[1] = 1;
HILL_HOLD := RX_3A0.DATA[2] = 1;
DISABLE_MCU_CAN := RX_3A0.DATA[3] = 1;
TRIP_RESET := RX_3A0.DATA[4] = 1;
BATTERY_CHARGING := RX_3A0.DATA[5] = 1;
DUMMY := RX_3A0.DATA[6] = 1;
(* Network 15 *)
TIMER_DATALOG(IN := RX_7F0.ERROR, PT := t#10s);
DATA_LOG_ERROR := TIMER_DATALOG.Q;
(* Network 16 *)
TIMER_DWIN(IN := RX_450.ERROR, PT := t#5s);
DWIN_CAN_ERROR := TIMER_DWIN.Q;
END_PROGRAM

(* POU FB_LIBRARY/RX_CAN, CFC *)
FUNCTION_BLOCK RX_CAN
(*
Created By: BHAGYESH
Date: 1-10-2023
Version: 1
Description: This function block checks the CAN data and updates the output CAN data only when it receives the new data.
*)
VAR_INPUT
	CHANNEL: BYTE;
	CAN_ID: DWORD;
END_VAR
VAR_OUTPUT
	DATA: ARRAY [0..7] OF BYTE;
	ERROR: BOOL;
END_VAR
VAR
	Rx: CAN_RX;

END_VAR
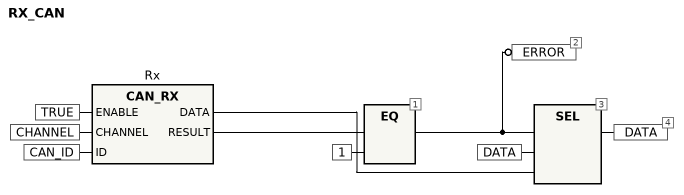
_CFC_ (* Continuous Function Chart, elements in execution order *)
#0 Rx:CAN_RX(ENABLE: TRUE, CHANNEL: CHANNEL, ID: CAN_ID)
#1 EQ(#0.RESULT, 1)
#2 ERROR <= NOT #1
#3 SEL(#1, DATA, #0.DATA)
#4 DATA <= #3
_END_CFC_
(* the same logic as Structured Text *)
Rx(ENABLE := TRUE, CHANNEL := CHANNEL, ID := CAN_ID);
ERROR := NOT (Rx.RESULT = 1);
DATA := SEL(Rx.RESULT = 1, DATA, Rx.DATA);
END_FUNCTION_BLOCK

(* POU FB_LIBRARY/PACK_BYTES, ST *)
FUNCTION_BLOCK PACK_BYTES
(*
Created by: Bhagyesh Unadkat
Date: 29-03-24
Version: 1
Updated by:
Update date:
Description: This block merges 8 bytes of data into 1 CAN data array.
*)
VAR_INPUT
	B0: BYTE;
	B1: BYTE;
	B2: BYTE;
	B3: BYTE;
	B4: BYTE;
	B5: BYTE;
	B6: BYTE;
	B7: BYTE;
END_VAR
VAR_OUTPUT
	CAN_DATA: ARRAY [0..7] OF BYTE;
END_VAR
CAN_DATA[0]:= B0;
CAN_DATA[1]:= B1;
CAN_DATA[2]:= B2;
CAN_DATA[3]:= B3;
CAN_DATA[4]:= B4;
CAN_DATA[5]:= B5;
CAN_DATA[6]:= B6;
CAN_DATA[7]:= B7;
END_FUNCTION_BLOCK

(* POU FB_LIBRARY/WORD_BYTE_CONVERSION, FBD *)
FUNCTION_BLOCK WORD_BYTE_CONVERSION
(*
Created by: Bhagyesh Unadkat
Date: 29-03-24
Version: 1
Updated by:
Update date:
Description: This block converts the WORD data into two BYTEs
*)
VAR_INPUT
	IN_WORD: WORD;
END_VAR
VAR_OUTPUT
	BYTE_H: BYTE;
	BYTE_L: BYTE;
END_VAR
VAR
END_VAR
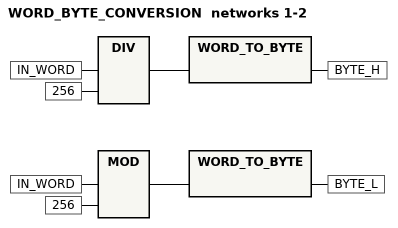
_FBD_ (* Function Block Diagram *)
NETWORK 1
	WORD_TO_BYTE(DIV(IN_WORD, 256)) => BYTE_H
NETWORK 2
	WORD_TO_BYTE(MOD(IN_WORD, 256)) => BYTE_L
_END_FBD_
(* the same logic as Structured Text *)
(* Network 1 *)
BYTE_H := WORD_TO_BYTE(IN_WORD / 256);
(* Network 2 *)
BYTE_L := WORD_TO_BYTE(IN_WORD MOD 256);
END_FUNCTION_BLOCK

(* POU FB_LIBRARY/DWORD_BYTE_CONVERSION, FBD *)
FUNCTION_BLOCK DWORD_BYTE_CONVERSION
(* BYTE_0 : LSB    ---------   BYTE_3 : MSB *)
VAR_INPUT
	INPUT_DWORD: DWORD;
END_VAR
VAR_OUTPUT
	BYTE_0: BYTE;
	BYTE_1: BYTE;
	BYTE_2: BYTE;
	BYTE_3: BYTE;
END_VAR
VAR
	WORD_1: WORD;
	WORD_2: WORD;
END_VAR
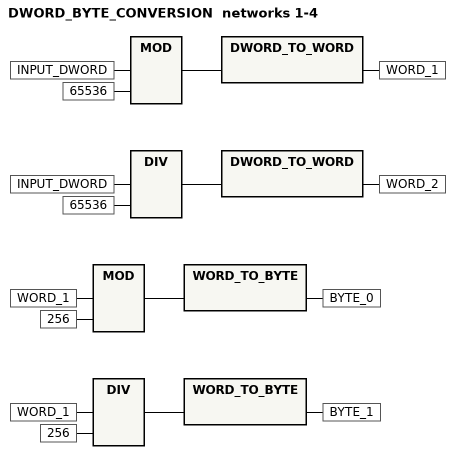
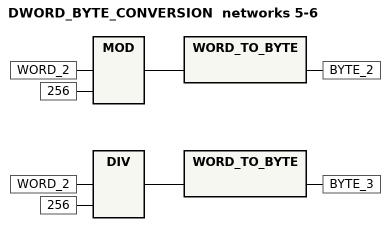
_FBD_ (* Function Block Diagram *)
NETWORK 1
	DWORD_TO_WORD(MOD(INPUT_DWORD, 65536)) => WORD_1
NETWORK 2
	DWORD_TO_WORD(DIV(INPUT_DWORD, 65536)) => WORD_2
NETWORK 3
	WORD_TO_BYTE(MOD(WORD_1, 256)) => BYTE_0
NETWORK 4
	WORD_TO_BYTE(DIV(WORD_1, 256)) => BYTE_1
NETWORK 5
	WORD_TO_BYTE(MOD(WORD_2, 256)) => BYTE_2
NETWORK 6
	WORD_TO_BYTE(DIV(WORD_2, 256)) => BYTE_3
_END_FBD_
(* the same logic as Structured Text *)
(* Network 1 *)
WORD_1 := DWORD_TO_WORD(INPUT_DWORD MOD 65536);
(* Network 2 *)
WORD_2 := DWORD_TO_WORD(INPUT_DWORD / 65536);
(* Network 3 *)
BYTE_0 := WORD_TO_BYTE(WORD_1 MOD 256);
(* Network 4 *)
BYTE_1 := WORD_TO_BYTE(WORD_1 / 256);
(* Network 5 *)
BYTE_2 := WORD_TO_BYTE(WORD_2 MOD 256);
(* Network 6 *)
BYTE_3 := WORD_TO_BYTE(WORD_2 / 256);
END_FUNCTION_BLOCK

(* POU CALCULATIONS, LD *)
PROGRAM CALCULATIONS
VAR
(*SPEED*)
	ABS_RPM1: INT;
	ABS_RPM2: INT;
	RPM_SUM: INT;
	AVG_RPM_REAL: REAL;
	SPEED_REAL: REAL;

(* RUNTIME*)
	MOTOR_1_RUNNING: BOOL;
	MOTOR_2_RUNNING: BOOL;
	HYDRAULIC_HOURS: BOOL;
	COUNT_HOURS: BOOL;
	RISE: R_TRIG;
	FALL: F_TRIG;

	PREVIOUS_TIME: REAL;
	HYDL_PREVIOUS_TIME: REAL;
	VEHICLE_PREVIOUS_TIME: REAL;
	VEHICLE_PREVIOUS_TIME_LT: REAL;

	TON_RUNTIME: TON;
	ET_REAL: REAL;
	HOURS_RUN: REAL;

(*ODO & TRIP*)
	INSTANTANEOUS_DISTANCE: REAL;
	TIMER_ODO: TON;
	ODO_KM_DWORD: DWORD;

(*RANGE*)
	ACTUAL_CAPACITY: REAL;
	ODO_TARGET: DWORD;
	ODO_CYCLE_COMPLETE: BOOL;
	OLD_CAPACITY: REAL;
	DIFFERENCE: REAL;
	CAPACITY_FACTOR: REAL;
	TIMER_RISING: TP;

	HOLD_PREVIOUS_VALUE: BOOL;
	INITIAL_RANGE_REAL: REAL;
	REMAINING_CAPACITY: INT;
	BATTERY1_REMAINING_CAPACITY: INT;
	BATTERY1_FULLCHARGE_HOURS: REAL;
	BATTERY2_REMAINING_CAPACITY: INT;
	BATTERY2_FULLCHARGE_HOURS: REAL;
	TON_HYDL_RUNTIME: TON;
	HYDL_HOURS_RUN: REAL;
	ET_REAL_HYDL: REAL;
	RISE_2: R_TRIG;
	FAL0_2L: F_TRIG;
	FALL_2: F_TRIG;
	ABS_RPM6: INT;
	MINUTE_RUN: REAL;
	ODO_TRIP: DWORD;
	ODO_TRIP_METER: DWORD;
	TRIP_KM_REAL: REAL;
	TRIP_DWORD_KM: DWORD;
	VEHICLE_UP_TIME_COUNT: BOOL;
	RISE_3: R_TRIG;
	FALL_3: F_TRIG;
	TON_VEHICLE_RUNTIME: TON;
	ET_REAL_VEHICLE: REAL;
	VEHICLE_HOURS_RUN: REAL;
	RISE_4: R_TRIG;
	FALL_4: F_TRIG;
	VEHICLE_UP_TIME_COUNT_BW: BOOL;
	VEHICLE_UP_TIME_COUNT_LT: BOOL;
	TON_VEHICLE_RUNTIME_LT: TON;
	ET_REAL_VEHICLE_LT: REAL;
	VEHICLE_HOURS_RUN_LT: REAL;
END_VAR
VAR CONSTANT
	METER_CYCLE: DWORD := 500;						(*CHANGES BASED ON THE CALCULATION OF DISTANCE FACTOR*)
	SPEED_FACTOR: REAL:= 0.00146726;
	ODO_DISTANCE_FACTOR: REAL:= 0.0002037860;	(*GLX with 72.02 Gear Ratio - 500ms Cycle time*)
	ODO_TIME: TIME := T#485MS;							(*Actual calculation factor is for 500ms*)
END_VAR
VAR RETAIN
	RETAIN_DISTANCE: REAL:=457860;							(*In meter*)(*28_03_25 *)
	RETAIN_TIME: REAL := 800640000;			(*222.4 hour- 28-03-25*)	(*Final: REAL:= 3600000 ; //1hour  = 3600000*)
	HYDL_RETAIN_TIME: REAL:=414640000;             (*114.9 HR*)
	VEHICLE_RETAIN_TIME: REAL:=2160000;
	VEHICLE_RETAIN_TIME_LT: REAL:= 801720000;  (*222.7*)
	SUBTRACT_TRIP: DWORD;

END_VAR
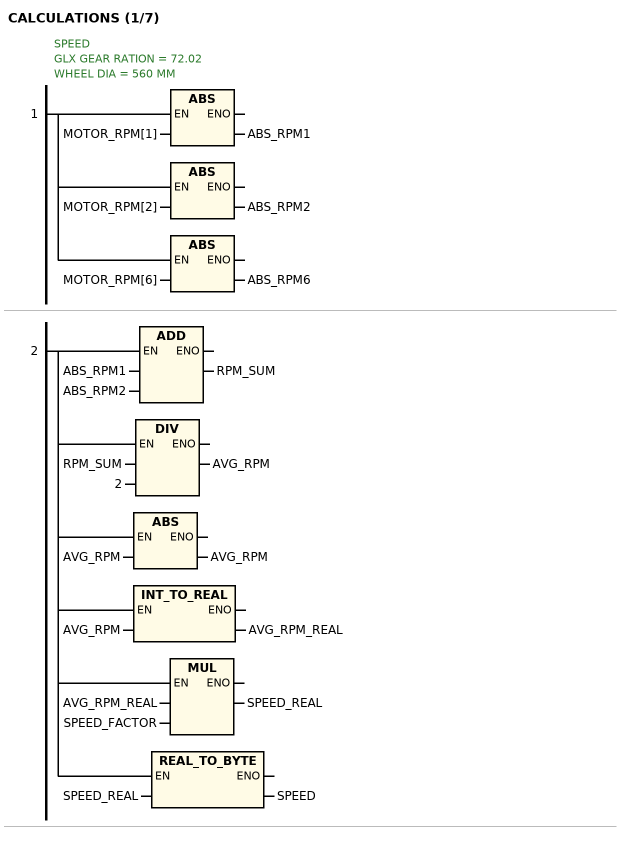
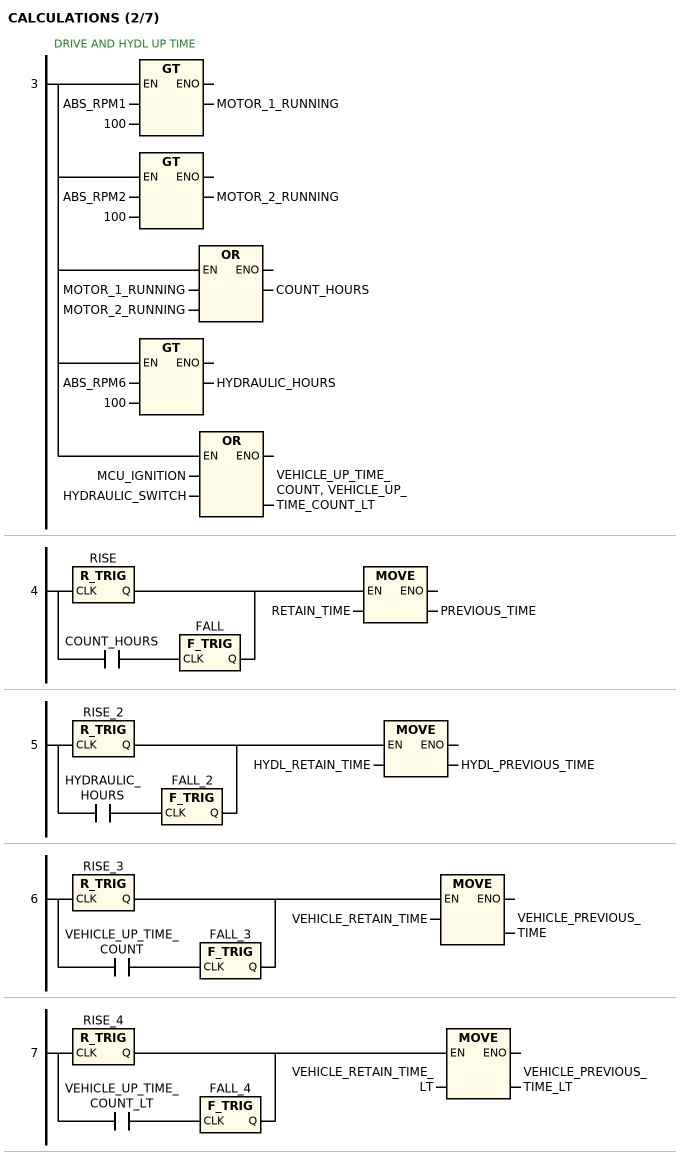
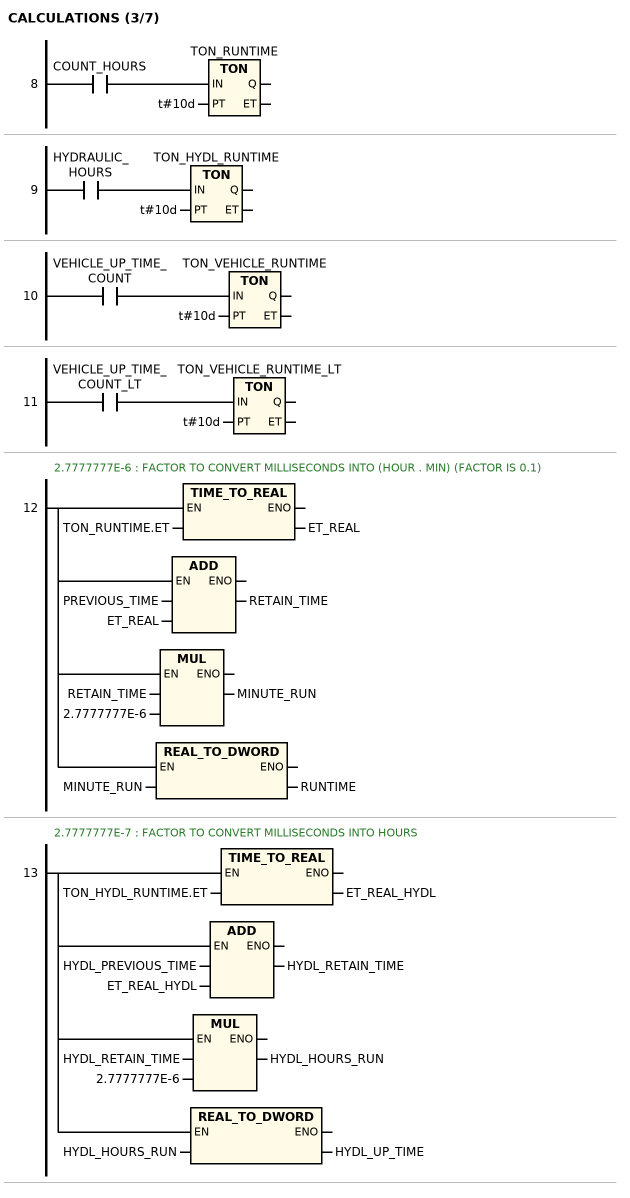
